			IF arrActualPrioInTurn[3] = 1 AND Lynus_Standards.GVL_Energy.stDataElectricHeatingElements[diNrOfEMS_OUT,liCounterCkeckDeviceAndPrio].byPriority = 1 AND
				(Lynus_Standards.GVL_Energy.stDataElectricHeatingElements[diNrOfEMS_OUT,liCounterCkeckDeviceAndPrio].arrTargetPowerEMS[1] <> 0 OR Lynus_Standards.GVL_Energy.stDataElectricHeatingElements[diNrOfEMS_OUT,liCounterCkeckDeviceAndPrio].arrTargetPowerEMS[2] <> 0 OR
					Lynus_Standards.GVL_Energy.stDataElectricHeatingElements[diNrOfEMS_OUT,liCounterCkeckDeviceAndPrio].arrTargetPowerEMS[3] <> 0 OR Lynus_Standards.GVL_Energy.stDataElectricHeatingElements[diNrOfEMS_OUT,liCounterCkeckDeviceAndPrio].arrTargetPowerEMS[4] <> 0 OR
						Lynus_Standards.GVL_Energy.stDataElectricHeatingElements[diNrOfEMS_OUT,liCounterCkeckDeviceAndPrio].arrTargetPowerEMS[5] <> 0 OR Lynus_Standards.GVL_Energy.stDataElectricHeatingElements[diNrOfEMS_OUT,liCounterCkeckDeviceAndPrio].arrTargetPowerEMS[6] <> 0 OR
							Lynus_Standards.GVL_Energy.stDataElectricHeatingElements[diNrOfEMS_OUT,liCounterCkeckDeviceAndPrio].arrTargetPowerEMS[7] <> 0 OR Lynus_Standards.GVL_Energy.stDataElectricHeatingElements[diNrOfEMS_OUT,liCounterCkeckDeviceAndPrio].arrTargetPowerEMS[8] <> 0 OR
								Lynus_Standards.GVL_Energy.stDataElectricHeatingElements[diNrOfEMS_OUT,liCounterCkeckDeviceAndPrio].arrTargetPowerEMS[9] <> 0 OR Lynus_Standards.GVL_Energy.stDataElectricHeatingElements[diNrOfEMS_OUT,liCounterCkeckDeviceAndPrio].arrTargetPowerEMS[10] <> 0) THEN 
									liNrOfNotDoneDevices := liNrOfNotDoneDevices + 1; 
			END_IF
				//1 Step
				IF arrActualPrioInTurn[3] = 255 AND Lynus_Standards.GVL_Energy.stDataElectricHeatingElements[diNrOfEMS_OUT,liCounterCkeckDeviceAndPrio].byPriority = 255 AND Lynus_Standards.GVL_Energy.stDataElectricHeatingElements[diNrOfEMS_OUT,liCounterCkeckDeviceAndPrio].byNumberOfSteps = 1 AND 
					Lynus_Standards.GVL_Energy.stDataElectricHeatingElements[diNrOfEMS_OUT,liCounterCkeckDeviceAndPrio].arrTargetPowerEMS[1] < 100 THEN 
						liNrOfNotDoneDevices := liNrOfNotDoneDevices + 1; 
				//2 Steps
				ELSIF arrActualPrioInTurn[3] = 255 AND Lynus_Standards.GVL_Energy.stDataElectricHeatingElements[diNrOfEMS_OUT,liCounterCkeckDeviceAndPrio].byPriority = 255 AND Lynus_Standards.GVL_Energy.stDataElectricHeatingElements[diNrOfEMS_OUT,liCounterCkeckDeviceAndPrio].byNumberOfSteps = 2 AND 
					(Lynus_Standards.GVL_Energy.stDataElectricHeatingElements[diNrOfEMS_OUT,liCounterCkeckDeviceAndPrio].arrTargetPowerEMS[1] < 100 OR Lynus_Standards.GVL_Energy.stDataElectricHeatingElements[diNrOfEMS_OUT,liCounterCkeckDeviceAndPrio].arrTargetPowerEMS[2] < 100) THEN 
						liNrOfNotDoneDevices := liNrOfNotDoneDevices + 1; 
				//3 Steps
				ELSIF arrActualPrioInTurn[3] = 255 AND Lynus_Standards.GVL_Energy.stDataElectricHeatingElements[diNrOfEMS_OUT,liCounterCkeckDeviceAndPrio].byPriority = 255 AND Lynus_Standards.GVL_Energy.stDataElectricHeatingElements[diNrOfEMS_OUT,liCounterCkeckDeviceAndPrio].byNumberOfSteps = 3 AND 
					(Lynus_Standards.GVL_Energy.stDataElectricHeatingElements[diNrOfEMS_OUT,liCounterCkeckDeviceAndPrio].arrTargetPowerEMS[1] < 100 OR Lynus_Standards.GVL_Energy.stDataElectricHeatingElements[diNrOfEMS_OUT,liCounterCkeckDeviceAndPrio].arrTargetPowerEMS[2] < 100 OR
						Lynus_Standards.GVL_Energy.stDataElectricHeatingElements[diNrOfEMS_OUT,liCounterCkeckDeviceAndPrio].arrTargetPowerEMS[3] < 100) THEN 
							liNrOfNotDoneDevices := liNrOfNotDoneDevices + 1;
				//4 Steps
				ELSIF arrActualPrioInTurn[3] = 255 AND Lynus_Standards.GVL_Energy.stDataElectricHeatingElements[diNrOfEMS_OUT,liCounterCkeckDeviceAndPrio].byPriority = 255 AND Lynus_Standards.GVL_Energy.stDataElectricHeatingElements[diNrOfEMS_OUT,liCounterCkeckDeviceAndPrio].byNumberOfSteps = 4 AND 
					(Lynus_Standards.GVL_Energy.stDataElectricHeatingElements[diNrOfEMS_OUT,liCounterCkeckDeviceAndPrio].arrTargetPowerEMS[1] < 100 OR Lynus_Standards.GVL_Energy.stDataElectricHeatingElements[diNrOfEMS_OUT,liCounterCkeckDeviceAndPrio].arrTargetPowerEMS[2] < 100 OR
						Lynus_Standards.GVL_Energy.stDataElectricHeatingElements[diNrOfEMS_OUT,liCounterCkeckDeviceAndPrio].arrTargetPowerEMS[3] < 100 OR Lynus_Standards.GVL_Energy.stDataElectricHeatingElements[diNrOfEMS_OUT,liCounterCkeckDeviceAndPrio].arrTargetPowerEMS[4] < 100) THEN 
							liNrOfNotDoneDevices := liNrOfNotDoneDevices + 1;  
				//5 Steps
				ELSIF arrActualPrioInTurn[3] = 255 AND Lynus_Standards.GVL_Energy.stDataElectricHeatingElements[diNrOfEMS_OUT,liCounterCkeckDeviceAndPrio].byPriority = 255 AND Lynus_Standards.GVL_Energy.stDataElectricHeatingElements[diNrOfEMS_OUT,liCounterCkeckDeviceAndPrio].byNumberOfSteps = 5 AND 
					(Lynus_Standards.GVL_Energy.stDataElectricHeatingElements[diNrOfEMS_OUT,liCounterCkeckDeviceAndPrio].arrTargetPowerEMS[1] < 100 OR Lynus_Standards.GVL_Energy.stDataElectricHeatingElements[diNrOfEMS_OUT,liCounterCkeckDeviceAndPrio].arrTargetPowerEMS[2] < 100 OR
						Lynus_Standards.GVL_Energy.stDataElectricHeatingElements[diNrOfEMS_OUT,liCounterCkeckDeviceAndPrio].arrTargetPowerEMS[3] < 100 OR Lynus_Standards.GVL_Energy.stDataElectricHeatingElements[diNrOfEMS_OUT,liCounterCkeckDeviceAndPrio].arrTargetPowerEMS[4] < 100 OR
							Lynus_Standards.GVL_Energy.stDataElectricHeatingElements[diNrOfEMS_OUT,liCounterCkeckDeviceAndPrio].arrTargetPowerEMS[5] < 100) THEN 
								liNrOfNotDoneDevices := liNrOfNotDoneDevices + 1; 
				//6 Steps
				ELSIF arrActualPrioInTurn[3] = 255 AND Lynus_Standards.GVL_Energy.stDataElectricHeatingElements[diNrOfEMS_OUT,liCounterCkeckDeviceAndPrio].byPriority = 255 AND Lynus_Standards.GVL_Energy.stDataElectricHeatingElements[diNrOfEMS_OUT,liCounterCkeckDeviceAndPrio].byNumberOfSteps = 6 AND 
					(Lynus_Standards.GVL_Energy.stDataElectricHeatingElements[diNrOfEMS_OUT,liCounterCkeckDeviceAndPrio].arrTargetPowerEMS[1] < 100 OR Lynus_Standards.GVL_Energy.stDataElectricHeatingElements[diNrOfEMS_OUT,liCounterCkeckDeviceAndPrio].arrTargetPowerEMS[2] < 100 OR
						Lynus_Standards.GVL_Energy.stDataElectricHeatingElements[diNrOfEMS_OUT,liCounterCkeckDeviceAndPrio].arrTargetPowerEMS[3] < 100 OR Lynus_Standards.GVL_Energy.stDataElectricHeatingElements[diNrOfEMS_OUT,liCounterCkeckDeviceAndPrio].arrTargetPowerEMS[4] < 100 OR
							Lynus_Standards.GVL_Energy.stDataElectricHeatingElements[diNrOfEMS_OUT,liCounterCkeckDeviceAndPrio].arrTargetPowerEMS[5] < 100 OR Lynus_Standards.GVL_Energy.stDataElectricHeatingElements[diNrOfEMS_OUT,liCounterCkeckDeviceAndPrio].arrTargetPowerEMS[6] < 100) THEN 
								liNrOfNotDoneDevices := liNrOfNotDoneDevices + 1; 
				//7 Steps
				ELSIF arrActualPrioInTurn[3] = 255 AND Lynus_Standards.GVL_Energy.stDataElectricHeatingElements[diNrOfEMS_OUT,liCounterCkeckDeviceAndPrio].byPriority = 255 AND Lynus_Standards.GVL_Energy.stDataElectricHeatingElements[diNrOfEMS_OUT,liCounterCkeckDeviceAndPrio].byNumberOfSteps = 7 AND 
					(Lynus_Standards.GVL_Energy.stDataElectricHeatingElements[diNrOfEMS_OUT,liCounterCkeckDeviceAndPrio].arrTargetPowerEMS[1] < 100 OR Lynus_Standards.GVL_Energy.stDataElectricHeatingElements[diNrOfEMS_OUT,liCounterCkeckDeviceAndPrio].arrTargetPowerEMS[2] < 100 OR
						Lynus_Standards.GVL_Energy.stDataElectricHeatingElements[diNrOfEMS_OUT,liCounterCkeckDeviceAndPrio].arrTargetPowerEMS[3] < 100 OR Lynus_Standards.GVL_Energy.stDataElectricHeatingElements[diNrOfEMS_OUT,liCounterCkeckDeviceAndPrio].arrTargetPowerEMS[4] < 100 OR
							Lynus_Standards.GVL_Energy.stDataElectricHeatingElements[diNrOfEMS_OUT,liCounterCkeckDeviceAndPrio].arrTargetPowerEMS[5] < 100 OR Lynus_Standards.GVL_Energy.stDataElectricHeatingElements[diNrOfEMS_OUT,liCounterCkeckDeviceAndPrio].arrTargetPowerEMS[6] < 100 OR
								Lynus_Standards.GVL_Energy.stDataElectricHeatingElements[diNrOfEMS_OUT,liCounterCkeckDeviceAndPrio].arrTargetPowerEMS[7] < 100) THEN 
									liNrOfNotDoneDevices := liNrOfNotDoneDevices + 1; 
				//8 Steps
				ELSIF arrActualPrioInTurn[3] = 255 AND Lynus_Standards.GVL_Energy.stDataElectricHeatingElements[diNrOfEMS_OUT,liCounterCkeckDeviceAndPrio].byPriority = 255 AND Lynus_Standards.GVL_Energy.stDataElectricHeatingElements[diNrOfEMS_OUT,liCounterCkeckDeviceAndPrio].byNumberOfSteps = 8 AND 
					(Lynus_Standards.GVL_Energy.stDataElectricHeatingElements[diNrOfEMS_OUT,liCounterCkeckDeviceAndPrio].arrTargetPowerEMS[1] < 100 OR Lynus_Standards.GVL_Energy.stDataElectricHeatingElements[diNrOfEMS_OUT,liCounterCkeckDeviceAndPrio].arrTargetPowerEMS[2] < 100 OR
						Lynus_Standards.GVL_Energy.stDataElectricHeatingElements[diNrOfEMS_OUT,liCounterCkeckDeviceAndPrio].arrTargetPowerEMS[3] < 100 OR Lynus_Standards.GVL_Energy.stDataElectricHeatingElements[diNrOfEMS_OUT,liCounterCkeckDeviceAndPrio].arrTargetPowerEMS[4] < 100 OR
							Lynus_Standards.GVL_Energy.stDataElectricHeatingElements[diNrOfEMS_OUT,liCounterCkeckDeviceAndPrio].arrTargetPowerEMS[5] < 100 OR Lynus_Standards.GVL_Energy.stDataElectricHeatingElements[diNrOfEMS_OUT,liCounterCkeckDeviceAndPrio].arrTargetPowerEMS[6] < 100 OR
								Lynus_Standards.GVL_Energy.stDataElectricHeatingElements[diNrOfEMS_OUT,liCounterCkeckDeviceAndPrio].arrTargetPowerEMS[7] < 100 OR Lynus_Standards.GVL_Energy.stDataElectricHeatingElements[diNrOfEMS_OUT,liCounterCkeckDeviceAndPrio].arrTargetPowerEMS[8] < 100) THEN 
									liNrOfNotDoneDevices := liNrOfNotDoneDevices + 1; 
				//9 Steps
				ELSIF arrActualPrioInTurn[3] = 255 AND Lynus_Standards.GVL_Energy.stDataElectricHeatingElements[diNrOfEMS_OUT,liCounterCkeckDeviceAndPrio].byPriority = 255 AND Lynus_Standards.GVL_Energy.stDataElectricHeatingElements[diNrOfEMS_OUT,liCounterCkeckDeviceAndPrio].byNumberOfSteps = 9 AND 
					(Lynus_Standards.GVL_Energy.stDataElectricHeatingElements[diNrOfEMS_OUT,liCounterCkeckDeviceAndPrio].arrTargetPowerEMS[1] < 100 OR Lynus_Standards.GVL_Energy.stDataElectricHeatingElements[diNrOfEMS_OUT,liCounterCkeckDeviceAndPrio].arrTargetPowerEMS[2] < 100 OR
						Lynus_Standards.GVL_Energy.stDataElectricHeatingElements[diNrOfEMS_OUT,liCounterCkeckDeviceAndPrio].arrTargetPowerEMS[3] < 100 OR Lynus_Standards.GVL_Energy.stDataElectricHeatingElements[diNrOfEMS_OUT,liCounterCkeckDeviceAndPrio].arrTargetPowerEMS[4] < 100 OR
							Lynus_Standards.GVL_Energy.stDataElectricHeatingElements[diNrOfEMS_OUT,liCounterCkeckDeviceAndPrio].arrTargetPowerEMS[5] < 100 OR Lynus_Standards.GVL_Energy.stDataElectricHeatingElements[diNrOfEMS_OUT,liCounterCkeckDeviceAndPrio].arrTargetPowerEMS[6] < 100 OR
								Lynus_Standards.GVL_Energy.stDataElectricHeatingElements[diNrOfEMS_OUT,liCounterCkeckDeviceAndPrio].arrTargetPowerEMS[7] < 100 OR Lynus_Standards.GVL_Energy.stDataElectricHeatingElements[diNrOfEMS_OUT,liCounterCkeckDeviceAndPrio].arrTargetPowerEMS[8] < 100 OR
									Lynus_Standards.GVL_Energy.stDataElectricHeatingElements[diNrOfEMS_OUT,liCounterCkeckDeviceAndPrio].arrTargetPowerEMS[9] < 100) THEN 
										liNrOfNotDoneDevices := liNrOfNotDoneDevices + 1; 
				//10 Steps
				ELSIF arrActualPrioInTurn[3] = 255 AND Lynus_Standards.GVL_Energy.stDataElectricHeatingElements[diNrOfEMS_OUT,liCounterCkeckDeviceAndPrio].byPriority = 255 AND Lynus_Standards.GVL_Energy.stDataElectricHeatingElements[diNrOfEMS_OUT,liCounterCkeckDeviceAndPrio].byNumberOfSteps = 10 AND 
					(Lynus_Standards.GVL_Energy.stDataElectricHeatingElements[diNrOfEMS_OUT,liCounterCkeckDeviceAndPrio].arrTargetPowerEMS[1] < 100 OR Lynus_Standards.GVL_Energy.stDataElectricHeatingElements[diNrOfEMS_OUT,liCounterCkeckDeviceAndPrio].arrTargetPowerEMS[2] < 100 OR
						Lynus_Standards.GVL_Energy.stDataElectricHeatingElements[diNrOfEMS_OUT,liCounterCkeckDeviceAndPrio].arrTargetPowerEMS[3] < 100 OR Lynus_Standards.GVL_Energy.stDataElectricHeatingElements[diNrOfEMS_OUT,liCounterCkeckDeviceAndPrio].arrTargetPowerEMS[4] < 100 OR
							Lynus_Standards.GVL_Energy.stDataElectricHeatingElements[diNrOfEMS_OUT,liCounterCkeckDeviceAndPrio].arrTargetPowerEMS[5] < 100 OR Lynus_Standards.GVL_Energy.stDataElectricHeatingElements[diNrOfEMS_OUT,liCounterCkeckDeviceAndPrio].arrTargetPowerEMS[6] < 100 OR
								Lynus_Standards.GVL_Energy.stDataElectricHeatingElements[diNrOfEMS_OUT,liCounterCkeckDeviceAndPrio].arrTargetPowerEMS[7] < 100 OR Lynus_Standards.GVL_Energy.stDataElectricHeatingElements[diNrOfEMS_OUT,liCounterCkeckDeviceAndPrio].arrTargetPowerEMS[8] < 100 OR
									Lynus_Standards.GVL_Energy.stDataElectricHeatingElements[diNrOfEMS_OUT,liCounterCkeckDeviceAndPrio].arrTargetPowerEMS[9] < 100 OR Lynus_Standards.GVL_Energy.stDataElectricHeatingElements[diNrOfEMS_OUT,liCounterCkeckDeviceAndPrio].arrTargetPowerEMS[10] < 100) THEN 
										liNrOfNotDoneDevices := liNrOfNotDoneDevices + 1; 
				END_IF
		
		IF arrActualPrioInTurn[3] = 1 AND uiState = 70 AND liNrOfNotDoneDevices = 0 AND arrCTCheckActivePrio[3] = Constants_Energy.diMaxNumberOfElectricHeatingElements AND liCounterCkeckDeviceAndPrio = Constants_Energy.diMaxNumberOfElectricHeatingElements THEN 
			arrMinPrioReached[3] := TRUE; arrMaxPrioReached[3] := FALSE; liNrOfNotDoneDevices := 0; uiState := 90; arrCTCheckActivePrio[3] := 0; liCounterCkeckDeviceAndPrio := 0; 
		END_IF
		IF arrActualPrioInTurn[3] = 255 AND uiState = 70 AND liNrOfNotDoneDevices = 0 AND arrCTCheckActivePrio[3] = Constants_Energy.diMaxNumberOfElectricHeatingElements AND liCounterCkeckDeviceAndPrio = Constants_Energy.diMaxNumberOfElectricHeatingElements THEN 
			arrMaxPrioReached[3] := TRUE; arrMinPrioReached[3] := FALSE; liNrOfNotDoneDevices := 0; uiState := 90; arrCTCheckActivePrio[3] := 0; liCounterCkeckDeviceAndPrio := 0; 
		END_IF
		
		//Timout, go to next step
		IF timTimeout.Q AND uiState = 70 THEN uiState := 90; END_IF
		
	90: //Check the priority for the big consumer to controll it
		uiState_CP := uiState;
	
		//First check if we have min 1 of this Device Type. If not, complete this Device Type and go to the next step
		//Check also the bigest Priority of this Device Type
		diNumberOfDevicesFromEachType := 0; bySearchBigestPrio := 0;
		FOR liLPCheckDeviceAndPrio := 1 TO Constants_Energy.diMaxNumberOfOtherBigConsumers BY 1 DO
			IF Lynus_Standards.GVL_Energy.stDataOtherBigConsumers[diNrOfEMS_OUT,liLPCheckDeviceAndPrio].byPriority <> 0 THEN diNumberOfDevicesFromEachType := diNumberOfDevicesFromEachType + 1; END_IF
				IF Lynus_Standards.GVL_Energy.stDataOtherBigConsumers[diNrOfEMS_OUT,liLPCheckDeviceAndPrio].byPriority > bySearchBigestPrio THEN bySearchBigestPrio := Lynus_Standards.GVL_Energy.stDataOtherBigConsumers[diNrOfEMS_OUT,liLPCheckDeviceAndPrio].byPriority; END_IF   
		END_FOR 
			IF bSurplusAvailable AND arrActualPrioInTurn[4] > bySearchBigestPrio AND uiState = 90 THEN arrActualPrioInTurn[4] := 255; END_IF
				IF NOT bSurplusAvailable AND arrActualPrioInTurn[4] > bySearchBigestPrio AND uiState = 90 THEN arrActualPrioInTurn[4] := bySearchBigestPrio; END_IF
		
			IF bSurplusAvailable AND diNumberOfDevicesFromEachType = 0 THEN arrActualPrioInTurn[4] := 255; END_IF
				IF NOT bSurplusAvailable AND diNumberOfDevicesFromEachType = 0 THEN arrActualPrioInTurn[4] := 1; END_IF
		
		//Count up each Device
		arrCTCheckActivePrio[4] := arrCTCheckActivePrio[4] + 1;
			arrCTCheckActivePrio[4] := LIMIT(1,arrCTCheckActivePrio[4],Constants_Energy.diMaxNumberOfOtherBigConsumers);
		
			//Surplus
			IF bSurplusAvailable AND Lynus_Standards.GVL_Energy.stDataOtherBigConsumers[diNrOfEMS_OUT,arrCTCheckActivePrio[4]].byPriority = arrActualPrioInTurn[4] AND Lynus_Standards.GVL_Energy.stDataOtherBigConsumers[diNrOfEMS_OUT,arrCTCheckActivePrio[4]].rTargetPowerEMS < 100 THEN
				arrMaxPrioReached[4] := FALSE;
					arrMinPrioReached[4] := FALSE;
						arrCTCheckActivePrio[4] := 0;
							uiState := 109; 
			ELSE
				IF bSurplusAvailable AND arrActualPrioInTurn[4] < 255 AND uiState = 90 AND arrCTCheckActivePrio[4] = Constants_Energy.diMaxNumberOfOtherBigConsumers THEN arrActualPrioInTurn[4] := arrActualPrioInTurn[4] + 1; arrCTCheckActivePrio[4] := 0; END_IF
			END_IF
				//No surplus
				IF NOT bSurplusAvailable AND Lynus_Standards.GVL_Energy.stDataOtherBigConsumers[diNrOfEMS_OUT,arrCTCheckActivePrio[4]].byPriority = arrActualPrioInTurn[4] AND Lynus_Standards.GVL_Energy.stDataOtherBigConsumers[diNrOfEMS_OUT,arrCTCheckActivePrio[4]].rTargetPowerEMS > 0 THEN
					arrMaxPrioReached[4] := FALSE;
						arrMinPrioReached[4] := FALSE;
							arrCTCheckActivePrio[4] := 0;
								uiState := 109;
				ELSE
					IF NOT bSurplusAvailable AND arrActualPrioInTurn[4] > 1 AND uiState = 90 AND arrCTCheckActivePrio[4] = Constants_Energy.diMaxNumberOfOtherBigConsumers THEN arrActualPrioInTurn[4] := arrActualPrioInTurn[4] - 1; arrCTCheckActivePrio[4] := 0; END_IF
				END_IF
		
		
		//Go to next step if we are on min prio or on max prio and the target power is just set to the min or to the max value.
		liNrOfNotDoneDevices := 0;
			FOR liLPCheckDeviceAndPrio := 1 TO Constants_Energy.diMaxNumberOfOtherBigConsumers BY 1 DO
				IF arrActualPrioInTurn[4] = 1 AND Lynus_Standards.GVL_Energy.stDataOtherBigConsumers[diNrOfEMS_OUT,liLPCheckDeviceAndPrio].rTargetPowerEMS <> 0 AND Lynus_Standards.GVL_Energy.stDataOtherBigConsumers[diNrOfEMS_OUT,liLPCheckDeviceAndPrio].byPriority = 1 THEN
					liNrOfNotDoneDevices := liNrOfNotDoneDevices + 1;	
				END_IF
					IF arrActualPrioInTurn[4] = 255 AND Lynus_Standards.GVL_Energy.stDataOtherBigConsumers[diNrOfEMS_OUT,liLPCheckDeviceAndPrio].rTargetPowerEMS < 100 AND Lynus_Standards.GVL_Energy.stDataOtherBigConsumers[diNrOfEMS_OUT,liLPCheckDeviceAndPrio].byPriority = 255 THEN
						liNrOfNotDoneDevices := liNrOfNotDoneDevices + 1;	
					END_IF
			END_FOR	
		
		IF arrActualPrioInTurn[4] = 1 AND uiState = 90 AND liNrOfNotDoneDevices = 0 AND arrCTCheckActivePrio[4] = Constants_Energy.diMaxNumberOfOtherBigConsumers THEN 
			arrMinPrioReached[4] := TRUE; arrMaxPrioReached[4] := FALSE; liNrOfNotDoneDevices := 0; uiState := 109; arrCTCheckActivePrio[4] := 0; 
		END_IF
		IF arrActualPrioInTurn[4] = 255 AND uiState = 90 AND liNrOfNotDoneDevices = 0 AND arrCTCheckActivePrio[4] = Constants_Energy.diMaxNumberOfOtherBigConsumers THEN 
			arrMaxPrioReached[4] := TRUE; arrMinPrioReached[4] := FALSE; liNrOfNotDoneDevices := 0; uiState := 109; arrCTCheckActivePrio[4] := 0; 
		END_IF
		
		//Timout, go to next step
		IF timTimeout.Q AND uiState = 90 THEN uiState := 109; END_IF
		
	109://Check if in Load management mode or Peak shaving mode some electric Fuse Line use to much power when we have here surplus
		uiState_CP := uiState;

		//Count up each Device
		arrCTCheckActivePrio[5] := arrCTCheckActivePrio[5] + 1;
			arrCTCheckActivePrio[5] := LIMIT(1,arrCTCheckActivePrio[5],Constants_Energy.diMaxNumberOfElectricChargingStations);
		
		IF ((eOperationMode = E_OperatingMode_EMS.eLoadManagement OR eOperationMode = E_OperatingMode_EMS.ePeakLoadCapping) AND bSurplusAvailable AND stSetupEMS.bEnableMainFuseFunction) THEN
			IF Lynus_Standards.GVL_Energy.stDataElectricChargingStations[diNrOfEMS_OUT,arrCTCheckActivePrio[5]].byPriority = arrActualPrioInTurn[5] THEN
				//The ECS use to much power. So dont give here more power. Go to next priority
				IF bNoPowerForECS THEN
					//Go to next prio that we can go forward with the other Devices with same priority. Controlling for ECS see down on the Part on wich we limit the charging station about the electric Fuse Line
					IF arrActualPrioInTurn[5] < 255 THEN arrActualPrioInTurn[5] := arrActualPrioInTurn[5] + 1; END_IF
						uiState := 110;
							arrCTCheckActivePrio[5] := 0;	
				END_IF
			END_IF 
		ELSE
			uiState := 110;
				arrCTCheckActivePrio[5] := 0;
		END_IF
		
		//Go to next step if wa have checked every ECS without resluts
		IF arrCTCheckActivePrio[5] >= Constants_Energy.diMaxNumberOfElectricChargingStations AND uiState = 109 THEN
			uiState := 110;
				arrCTCheckActivePrio[5] := 0;
		END_IF 
	 	
		//Timout, go to next step
		IF timTimeout.Q AND uiState = 109 THEN uiState := 110; arrCTCheckActivePrio[5] := 0; END_IF	
		
	110: //Check the priority for the electric charging stations to controll it
		uiState_CP := uiState;
	
		//First check if we have min 1 of this Device Type. If not, complete this Device Type and go to the next step
		//Check also the bigest Priority of this Device Type
		diNumberOfDevicesFromEachType := 0; bySearchBigestPrio := 0;
		FOR liLPCheckDeviceAndPrio := 1 TO Constants_Energy.diMaxNumberOfElectricChargingStations BY 1 DO
			IF Lynus_Standards.GVL_Energy.stDataElectricChargingStations[diNrOfEMS_OUT,liLPCheckDeviceAndPrio].byPriority <> 0 THEN diNumberOfDevicesFromEachType := diNumberOfDevicesFromEachType + 1; END_IF
				IF Lynus_Standards.GVL_Energy.stDataElectricChargingStations[diNrOfEMS_OUT,liLPCheckDeviceAndPrio].byPriority > bySearchBigestPrio THEN bySearchBigestPrio := Lynus_Standards.GVL_Energy.stDataElectricChargingStations[diNrOfEMS_OUT,liLPCheckDeviceAndPrio].byPriority; END_IF   
		END_FOR 
			IF bSurplusAvailable AND arrActualPrioInTurn[5] > bySearchBigestPrio AND uiState = 110 THEN arrActualPrioInTurn[5] := 255; END_IF
				IF NOT bSurplusAvailable AND arrActualPrioInTurn[5] > bySearchBigestPrio AND uiState = 110 THEN arrActualPrioInTurn[5] := bySearchBigestPrio; END_IF
		
			IF bSurplusAvailable AND diNumberOfDevicesFromEachType = 0 THEN arrActualPrioInTurn[5] := 255; END_IF
				IF NOT bSurplusAvailable AND diNumberOfDevicesFromEachType = 0 THEN arrActualPrioInTurn[5] := 1; END_IF
		
		//Count up each Device
		arrCTCheckActivePrio[5] := arrCTCheckActivePrio[5] + 1;
			arrCTCheckActivePrio[5] := LIMIT(1,arrCTCheckActivePrio[5],Constants_Energy.diMaxNumberOfElectricChargingStations);
		
			//Surplus
			IF bSurplusAvailable AND Lynus_Standards.GVL_Energy.stDataElectricChargingStations[diNrOfEMS_OUT,arrCTCheckActivePrio[5]].byPriority = arrActualPrioInTurn[5] AND Lynus_Standards.GVL_Energy.stDataElectricChargingStations[diNrOfEMS_OUT,arrCTCheckActivePrio[5]].rTargetPowerEMS < 100 THEN
				arrMaxPrioReached[5] := FALSE;
					arrMinPrioReached[5] := FALSE;
						arrCTCheckActivePrio[5] := 0;
							uiState := 130;
			ELSE
				IF bSurplusAvailable AND arrActualPrioInTurn[5] < 255 AND uiState = 110 AND arrCTCheckActivePrio[5] = Constants_Energy.diMaxNumberOfElectricChargingStations THEN arrActualPrioInTurn[5] := arrActualPrioInTurn[5] + 1; arrCTCheckActivePrio[5] := 0; END_IF
			END_IF
				//No surplus
				IF NOT bSurplusAvailable AND Lynus_Standards.GVL_Energy.stDataElectricChargingStations[diNrOfEMS_OUT,arrCTCheckActivePrio[5]].byPriority = arrActualPrioInTurn[5] AND Lynus_Standards.GVL_Energy.stDataElectricChargingStations[diNrOfEMS_OUT,arrCTCheckActivePrio[5]].rTargetPowerEMS > 0 THEN
					arrMaxPrioReached[5] := FALSE;
						arrMinPrioReached[5] := FALSE;
							arrCTCheckActivePrio[5] := 0;
								uiState := 130;
				ELSE
					IF NOT bSurplusAvailable AND arrActualPrioInTurn[5] > 1 AND uiState = 110 AND arrCTCheckActivePrio[5] = Constants_Energy.diMaxNumberOfElectricChargingStations THEN arrActualPrioInTurn[5] := arrActualPrioInTurn[5] - 1; arrCTCheckActivePrio[5] := 0; END_IF
				END_IF
		
		//Go to next step if we are on min prio or on max prio and the target power is just set to the min or to the max value.
		liNrOfNotDoneDevices := 0;
			FOR liLPCheckDeviceAndPrio := 1 TO Constants_Energy.diMaxNumberOfElectricChargingStations BY 1 DO
				IF arrActualPrioInTurn[5] = 1 AND Lynus_Standards.GVL_Energy.stDataElectricChargingStations[diNrOfEMS_OUT,liLPCheckDeviceAndPrio].rTargetPowerEMS <> 0 AND Lynus_Standards.GVL_Energy.stDataElectricChargingStations[diNrOfEMS_OUT,liLPCheckDeviceAndPrio].byPriority = 1 THEN
					liNrOfNotDoneDevices := liNrOfNotDoneDevices + 1;	
				END_IF
					IF arrActualPrioInTurn[5] = 255 AND Lynus_Standards.GVL_Energy.stDataElectricChargingStations[diNrOfEMS_OUT,liLPCheckDeviceAndPrio].rTargetPowerEMS < 100 AND Lynus_Standards.GVL_Energy.stDataElectricChargingStations[diNrOfEMS_OUT,liLPCheckDeviceAndPrio].byPriority = 255 THEN
						liNrOfNotDoneDevices := liNrOfNotDoneDevices + 1;	
					END_IF
			END_FOR
		
		IF arrActualPrioInTurn[5] = 1 AND uiState = 110 AND liNrOfNotDoneDevices = 0 AND arrCTCheckActivePrio[5] = Constants_Energy.diMaxNumberOfElectricChargingStations THEN 
			arrMinPrioReached[5] := TRUE; arrMaxPrioReached[5] := FALSE; liNrOfNotDoneDevices := 0; uiState := 130; arrCTCheckActivePrio[5] := 0; 
		END_IF
		IF arrActualPrioInTurn[5] = 255 AND uiState = 110 AND liNrOfNotDoneDevices = 0 AND arrCTCheckActivePrio[5] = Constants_Energy.diMaxNumberOfElectricChargingStations THEN 
			arrMaxPrioReached[5] := TRUE; arrMinPrioReached[5] := FALSE; liNrOfNotDoneDevices := 0; uiState := 130; arrCTCheckActivePrio[5] := 0; 
		END_IF	
		
		//Timout, go to next step
		IF timTimeout.Q AND uiState = 110 THEN uiState := 130; END_IF
		
	130: //Search the smallest/biggest common priority and the number of devices with the same priority  
		IF bSurplusAvailable THEN bySmGrActiveCommonPrio := 255; END_IF
		IF NOT bSurplusAvailable THEN bySmGrActiveCommonPrio := 1; END_IF
	
		FOR byLPSmActiveCommonPrio := 1 TO 5 BY 1 DO
			IF bSurplusAvailable AND arrActualPrioInTurn[byLPSmActiveCommonPrio] < bySmGrActiveCommonPrio THEN bySmGrActiveCommonPrio := arrActualPrioInTurn[byLPSmActiveCommonPrio]; END_IF 
			IF NOT bSurplusAvailable AND arrActualPrioInTurn[byLPSmActiveCommonPrio] > bySmGrActiveCommonPrio THEN bySmGrActiveCommonPrio := arrActualPrioInTurn[byLPSmActiveCommonPrio]; END_IF 
		END_FOR
		
		//Back to the start when complete power is awarded, all power is set on 0 or we haven't common priority 	
		IF (arrMaxPrioReached[1] AND arrMaxPrioReached[2] AND arrMaxPrioReached[3] AND arrMaxPrioReached[4] AND arrMaxPrioReached[5]) OR
			(arrMinPrioReached[1] AND arrMinPrioReached[2] AND arrMinPrioReached[3] AND arrMinPrioReached[4] AND arrMinPrioReached[5]) THEN
				uiState := 10;
		ELSE
				uiState := 131;
		END_IF
		
	131: //Ckeck if the Batterys are full or not when we have no surplus. Thus the problem can be avoided if the battery FB regulates the power internally to 0, but the EMS still sends power to the inverter.
		 //Because otherwise it always takes too long when we have a small consumption and the battery must first be regulated to 0% in the GVL, although you are already full and you can therefore no longer be regulated back.
		 
		IF eOperationMode = E_OperatingMode_EMS.eSelfConsumption THEN 
			FOR liLPDataBatteryInverter := 1 TO Constants_Energy.diMaxNumberOfBatteryInverters BY 1 DO
				IF NOT bSurplusAvailable AND Lynus_Standards.GVL_Energy.stDataOfBatteryInverters[diNrOfEMS_OUT,liLPDataBatteryInverter].byPriority = bySmGrActiveCommonPrio AND 
					arrTimBatterysAreFull[liLPDataBatteryInverter].Q THEN
						Lynus_Standards.GVL_Energy.stDataOfBatteryInverters[diNrOfEMS_OUT,liLPDataBatteryInverter].rTargetPowerEMS := 0;
				END_IF	  
			END_FOR 
	
			//When we have a surplus again and the battery is full, we control it again with - 99.99%, so that the following devices do not have to wait too long to be controlled. 	
			//It must be set to 99.99, otherwise an error would occur in the next step.
			FOR liLPDataBatteryInverter := 1 TO Constants_Energy.diMaxNumberOfBatteryInverters BY 1 DO
				IF bSurplusAvailable AND Lynus_Standards.GVL_Energy.stDataOfBatteryInverters[diNrOfEMS_OUT,liLPDataBatteryInverter].byPriority = bySmGrActiveCommonPrio AND 
					arrTimBatterysAreFull[liLPDataBatteryInverter].Q THEN
						Lynus_Standards.GVL_Energy.stDataOfBatteryInverters[diNrOfEMS_OUT,liLPDataBatteryInverter].rTargetPowerEMS := - 99.99;
				END_IF	  
			END_FOR
		END_IF
		
		//Go to the next Step
		uiState := 150;
		
	150: //Calcualte the % power from each device with the same priority
		lrMaxPowerDevicesWithActualPrio := 0;
			bMissingPowerData := FALSE;
		
		//Batterys are only a "normal" Device, when the self consumption mode is active.
		IF eOperationMode = E_OperatingMode_EMS.eSelfConsumption THEN 
			//Batteryinverters
			FOR liLPCheckMaxPower := 1 TO Constants_Energy.diMaxNumberOfBatteryInverters BY 1 DO
				IF bSurplusAvailable AND Lynus_Standards.GVL_Energy.stDataOfBatteryInverters[diNrOfEMS_OUT,liLPCheckMaxPower].byPriority = bySmGrActiveCommonPrio AND Lynus_Standards.GVL_Energy.stDataOfBatteryInverters[diNrOfEMS_OUT,liLPCheckMaxPower].rTargetPowerEMS > -100 AND NOT Lynus_Standards.GVL_Energy.stDataOfBatteryInverters[diNrOfEMS_OUT,liLPCheckMaxPower].bWorkOnIslandMode THEN lrMaxPowerDevicesWithActualPrio := lrMaxPowerDevicesWithActualPrio + Lynus_Standards.GVL_Energy.stDataOfBatteryInverters[diNrOfEMS_OUT,liLPCheckMaxPower].rMaxChargePower; END_IF
				IF NOT bSurplusAvailable AND Lynus_Standards.GVL_Energy.stDataOfBatteryInverters[diNrOfEMS_OUT,liLPCheckMaxPower].byPriority = bySmGrActiveCommonPrio AND Lynus_Standards.GVL_Energy.stDataOfBatteryInverters[diNrOfEMS_OUT,liLPCheckMaxPower].rTargetPowerEMS < 0 AND NOT Lynus_Standards.GVL_Energy.stDataOfBatteryInverters[diNrOfEMS_OUT,liLPCheckMaxPower].bWorkOnIslandMode THEN lrMaxPowerDevicesWithActualPrio := lrMaxPowerDevicesWithActualPrio + Lynus_Standards.GVL_Energy.stDataOfBatteryInverters[diNrOfEMS_OUT,liLPCheckMaxPower].rMaxChargePower; END_IF 
			END_FOR
		END_IF
			//Heating pumps
			IF arrActualStepInTurn[1] >= 1 AND arrActualStepInTurn[1] <= 2 THEN
				FOR liLPCheckMaxPower := 1 TO Constants_Energy.diMaxNumberOfHeatingPumps BY 1 DO
					IF bSurplusAvailable AND Lynus_Standards.GVL_Energy.stDataHeatingPumps[diNrOfEMS_OUT,liLPCheckMaxPower].byPriority = bySmGrActiveCommonPrio AND Lynus_Standards.GVL_Energy.stDataHeatingPumps[diNrOfEMS_OUT,liLPCheckMaxPower].arrTargetPowerEMS[arrActualStepInTurn[1]] < 100 THEN lrMaxPowerDevicesWithActualPrio := lrMaxPowerDevicesWithActualPrio + Lynus_Standards.GVL_Energy.stDataHeatingPumps[diNrOfEMS_OUT,liLPCheckMaxPower].arrMaxPower[arrActualStepInTurn[1]]; END_IF
					IF NOT bSurplusAvailable AND Lynus_Standards.GVL_Energy.stDataHeatingPumps[diNrOfEMS_OUT,liLPCheckMaxPower].byPriority = bySmGrActiveCommonPrio AND Lynus_Standards.GVL_Energy.stDataHeatingPumps[diNrOfEMS_OUT,liLPCheckMaxPower].arrTargetPowerEMS[arrActualStepInTurn[1]] > 0 THEN lrMaxPowerDevicesWithActualPrio := lrMaxPowerDevicesWithActualPrio + Lynus_Standards.GVL_Energy.stDataHeatingPumps[diNrOfEMS_OUT,liLPCheckMaxPower].arrMaxPower[arrActualStepInTurn[1]]; END_IF
				END_FOR
			END_IF
				//Electric heating elements
				IF arrActualStepInTurn[2] >= 1 AND arrActualStepInTurn[2] <= 10 THEN
					FOR liLPCheckMaxPower := 1 TO Constants_Energy.diMaxNumberOfElectricHeatingElements BY 1 DO
						IF bSurplusAvailable AND Lynus_Standards.GVL_Energy.stDataElectricHeatingElements[diNrOfEMS_OUT,liLPCheckMaxPower].byPriority = bySmGrActiveCommonPrio AND Lynus_Standards.GVL_Energy.stDataElectricHeatingElements[diNrOfEMS_OUT,liLPCheckMaxPower].arrTargetPowerEMS[arrActualStepInTurn[2]] < 100 THEN lrMaxPowerDevicesWithActualPrio := lrMaxPowerDevicesWithActualPrio + Lynus_Standards.GVL_Energy.stDataElectricHeatingElements[diNrOfEMS_OUT,liLPCheckMaxPower].arrMaxPower[arrActualStepInTurn[2]]; END_IF 
						IF NOT bSurplusAvailable AND Lynus_Standards.GVL_Energy.stDataElectricHeatingElements[diNrOfEMS_OUT,liLPCheckMaxPower].byPriority = bySmGrActiveCommonPrio AND Lynus_Standards.GVL_Energy.stDataElectricHeatingElements[diNrOfEMS_OUT,liLPCheckMaxPower].arrTargetPowerEMS[arrActualStepInTurn[2]] > 0 THEN lrMaxPowerDevicesWithActualPrio := lrMaxPowerDevicesWithActualPrio + Lynus_Standards.GVL_Energy.stDataElectricHeatingElements[diNrOfEMS_OUT,liLPCheckMaxPower].arrMaxPower[arrActualStepInTurn[2]]; END_IF 
					END_FOR	
				END_IF
					//Other big consumer
					FOR liLPCheckMaxPower := 1 TO Constants_Energy.diMaxNumberOfOtherBigConsumers BY 1 DO
						IF bSurplusAvailable AND Lynus_Standards.GVL_Energy.stDataOtherBigConsumers[diNrOfEMS_OUT,liLPCheckMaxPower].byPriority = bySmGrActiveCommonPrio AND Lynus_Standards.GVL_Energy.stDataOtherBigConsumers[diNrOfEMS_OUT,liLPCheckMaxPower].rTargetPowerEMS < 100 THEN lrMaxPowerDevicesWithActualPrio := lrMaxPowerDevicesWithActualPrio + Lynus_Standards.GVL_Energy.stDataOtherBigConsumers[diNrOfEMS_OUT,liLPCheckMaxPower].rMaxPower; END_IF
						IF NOT bSurplusAvailable AND Lynus_Standards.GVL_Energy.stDataOtherBigConsumers[diNrOfEMS_OUT,liLPCheckMaxPower].byPriority = bySmGrActiveCommonPrio AND Lynus_Standards.GVL_Energy.stDataOtherBigConsumers[diNrOfEMS_OUT,liLPCheckMaxPower].rTargetPowerEMS > 0 THEN lrMaxPowerDevicesWithActualPrio := lrMaxPowerDevicesWithActualPrio + Lynus_Standards.GVL_Energy.stDataOtherBigConsumers[diNrOfEMS_OUT,liLPCheckMaxPower].rMaxPower; END_IF
					END_FOR
						//Electric charging stations
						FOR liLPCheckMaxPower := 1 TO Constants_Energy.diMaxNumberOfElectricChargingStations BY 1 DO
							IF bSurplusAvailable AND Lynus_Standards.GVL_Energy.stDataElectricChargingStations[diNrOfEMS_OUT,liLPCheckMaxPower].byPriority = bySmGrActiveCommonPrio AND Lynus_Standards.GVL_Energy.stDataElectricChargingStations[diNrOfEMS_OUT,liLPCheckMaxPower].rTargetPowerEMS < 100 THEN lrMaxPowerDevicesWithActualPrio := lrMaxPowerDevicesWithActualPrio + Lynus_Standards.GVL_Energy.stDataElectricChargingStations[diNrOfEMS_OUT,liLPCheckMaxPower].rMaxPower; END_IF
							IF NOT bSurplusAvailable AND Lynus_Standards.GVL_Energy.stDataElectricChargingStations[diNrOfEMS_OUT,liLPCheckMaxPower].byPriority = bySmGrActiveCommonPrio AND Lynus_Standards.GVL_Energy.stDataElectricChargingStations[diNrOfEMS_OUT,liLPCheckMaxPower].rTargetPowerEMS > 0 THEN lrMaxPowerDevicesWithActualPrio := lrMaxPowerDevicesWithActualPrio + Lynus_Standards.GVL_Energy.stDataElectricChargingStations[diNrOfEMS_OUT,liLPCheckMaxPower].rMaxPower; END_IF 
						END_FOR
		
		//Check is somthing has changed at the actual priority or at the actual step 
		//Priority or step now is higher as before
		IF (bSurplusAvailable AND MEMCMP(ADR(bySmGrActiveCommonPrio),ADR(bySmGrActiveCommonPrio_CP),SIZEOF(bySmGrActiveCommonPrio_CP)) <> 0) OR (bSurplusAvailable AND MEMCMP(ADR(arrActualStepInTurn),ADR(arrActualStepInTurn_CP),SIZEOF(arrActualStepInTurn_CP)) <> 0) THEN
			bySmGrActiveCommonPrio_CP := bySmGrActiveCommonPrio;
				arrActualStepInTurn_CP := arrActualStepInTurn;
					bStepWasOn100 := FALSE;		
		END_IF
			//Priority or step now is lower as before
			IF (NOT bSurplusAvailable AND MEMCMP(ADR(bySmGrActiveCommonPrio),ADR(bySmGrActiveCommonPrio_CP),SIZEOF(bySmGrActiveCommonPrio_CP)) <> 0) OR (NOT bSurplusAvailable AND MEMCMP(ADR(arrActualStepInTurn),ADR(arrActualStepInTurn_CP),SIZEOF(arrActualStepInTurn_CP)) <> 0) THEN
				bySmGrActiveCommonPrio_CP := bySmGrActiveCommonPrio;
					arrActualStepInTurn_CP := arrActualStepInTurn;
						bStepWasOn100 := TRUE;			
			END_IF						
						
		IF lrMaxPowerDevicesWithActualPrio > 0 THEN
			//Calcualte the power for the controllable devices
			IF bSurplusAvailable THEN rValuePercentToControllableDevices := LREAL_TO_REAL((100 * (lrActualSurplusOrConsumption * - 1)) / lrMaxPowerDevicesWithActualPrio); END_IF
  			IF NOT bSurplusAvailable THEN rValuePercentToControllableDevices := LREAL_TO_REAL((100 * lrActualSurplusOrConsumption) / lrMaxPowerDevicesWithActualPrio); END_IF
			//Calcualte the power for the On/Off or step switched devices
			IF bSurplusAvailable THEN rValuePercentToStepSwitchedDevices := LREAL_TO_REAL((100 * (lrActualSurplusOrConsumption * - 1)) / lrMaxPowerDevicesWithActualPrio); END_IF
			IF NOT bSurplusAvailable THEN rValuePercentToStepSwitchedDevices := (100 - LREAL_TO_REAL((100 * lrActualSurplusOrConsumption) / lrMaxPowerDevicesWithActualPrio)); END_IF
				IF bSurplusAvailable AND rValuePercentToStepSwitchedDevices >= 100 THEN bStepWasOn100 := TRUE; END_IF
				IF NOT bSurplusAvailable AND rValuePercentToStepSwitchedDevices < Constants_Energy.byTargetOffPowerForOnOffDevices THEN bStepWasOn100 := FALSE; END_IF
					IF bStepWasOn100 THEN rValuePercentToStepSwitchedDevices := 100; END_IF
					IF NOT bStepWasOn100 THEN rValuePercentToStepSwitchedDevices := 0; END_IF		
		ELSE
			//Power inputs from the setups of the devices are missing. Set the target power automatically to 0
			bMissingPowerData := TRUE;
			IF bSurplusAvailable THEN
				rValuePercentToControllableDevices := - 100;
				rValuePercentToStepSwitchedDevices := 0;
			END_IF
				IF NOT bSurplusAvailable THEN
					rValuePercentToControllableDevices := 100;
					rValuePercentToStepSwitchedDevices := 0;
				END_IF
		END_IF
		
		//If we have more surplus than the maximum power of the devices is, then we can set the target power directly to 100%
		IF bSurplusAvailable AND (lrActualSurplusOrConsumption * - 1) >= lrMaxPowerDevicesWithActualPrio AND NOT bMissingPowerData THEN rValuePercentToControllableDevices := 100; END_IF
		IF bSurplusAvailable AND (lrActualSurplusOrConsumption * - 1) >= lrMaxPowerDevicesWithActualPrio AND NOT bMissingPowerData THEN rValuePercentToStepSwitchedDevices := 100; bStepWasOn100 := TRUE; END_IF
		
		//If more power is consumed than the maximum power of the devices, 0% power can be commanded (for controllable devices 100% as it is deducted).
		IF NOT bSurplusAvailable AND lrActualSurplusOrConsumption >= lrMaxPowerDevicesWithActualPrio AND NOT bMissingPowerData THEN rValuePercentToControllableDevices := 100; END_IF
		IF NOT bSurplusAvailable AND lrActualSurplusOrConsumption >= lrMaxPowerDevicesWithActualPrio AND NOT bMissingPowerData THEN rValuePercentToStepSwitchedDevices := 0; bStepWasOn100 := FALSE; END_IF
		
		//Check the limits
		rValuePercentToControllableDevices := LIMIT(0,rValuePercentToControllableDevices,100);
			rValuePercentToStepSwitchedDevices := LIMIT(0,rValuePercentToStepSwitchedDevices,100);
				
		uiState := 170;
		
	170: //Set the target power to each device
		//Batterys or battery inverters
		//Batterys are only a "normal" Device, when the self consumption mode is active.
		IF eOperationMode = E_OperatingMode_EMS.eSelfConsumption THEN 
			FOR liLPSetPercentPower := 1 TO Constants_Energy.diMaxNumberOfBatteryInverters BY 1 DO
				IF bSurplusAvailable AND Lynus_Standards.GVL_Energy.stDataOfBatteryInverters[diNrOfEMS_OUT,liLPSetPercentPower].byPriority = bySmGrActiveCommonPrio AND Lynus_Standards.GVL_Energy.stDataOfBatteryInverters[diNrOfEMS_OUT,liLPSetPercentPower].rTargetPowerEMS > -100 THEN 
					Lynus_Standards.GVL_Energy.stDataOfBatteryInverters[diNrOfEMS_OUT,liLPSetPercentPower].rTargetPowerEMS := Lynus_Standards.GVL_Energy.stDataOfBatteryInverters[diNrOfEMS_OUT,liLPSetPercentPower].rTargetPowerEMS - rValuePercentToControllableDevices; 
				END_IF
				IF bSurplusAvailable AND Lynus_Standards.GVL_Energy.stDataOfBatteryInverters[diNrOfEMS_OUT,liLPSetPercentPower].rTargetPowerEMS < -100 THEN 
					Lynus_Standards.GVL_Energy.stDataOfBatteryInverters[diNrOfEMS_OUT,liLPSetPercentPower].rTargetPowerEMS := -100; 
				END_IF 
				IF NOT bSurplusAvailable AND Lynus_Standards.GVL_Energy.stDataOfBatteryInverters[diNrOfEMS_OUT,liLPSetPercentPower].byPriority = bySmGrActiveCommonPrio AND Lynus_Standards.GVL_Energy.stDataOfBatteryInverters[diNrOfEMS_OUT,liLPSetPercentPower].rTargetPowerEMS < 0 THEN 
					Lynus_Standards.GVL_Energy.stDataOfBatteryInverters[diNrOfEMS_OUT,liLPSetPercentPower].rTargetPowerEMS := Lynus_Standards.GVL_Energy.stDataOfBatteryInverters[diNrOfEMS_OUT,liLPSetPercentPower].rTargetPowerEMS + rValuePercentToControllableDevices;
				
				END_IF
				IF NOT bSurplusAvailable AND Lynus_Standards.GVL_Energy.stDataOfBatteryInverters[diNrOfEMS_OUT,liLPSetPercentPower].rTargetPowerEMS > 0 THEN 
					Lynus_Standards.GVL_Energy.stDataOfBatteryInverters[diNrOfEMS_OUT,liLPSetPercentPower].rTargetPowerEMS := 0;
					
				END_IF
				//Power Data is Missing
				IF bMissingPowerData AND Lynus_Standards.GVL_Energy.stDataOfBatteryInverters[diNrOfEMS_OUT,liLPSetPercentPower].byPriority = bySmGrActiveCommonPrio THEN 
					Lynus_Standards.GVL_Energy.stDataOfBatteryInverters[diNrOfEMS_OUT,liLPSetPercentPower].rTargetPowerEMS := 0;	
				END_IF 
				//Limit
							Lynus_Standards.GVL_Energy.stDataOfBatteryInverters[diNrOfEMS_OUT,liLPSetPercentPower].rTargetPowerEMS := LIMIT(-100,Lynus_Standards.GVL_Energy.stDataOfBatteryInverters[diNrOfEMS_OUT,liLPSetPercentPower].rTargetPowerEMS,100);	
			END_FOR
		END_IF
			//Heating pumps
			IF arrActualStepInTurn[1] >= 1 AND arrActualStepInTurn[1] <= 2 THEN
				FOR liLPSetPercentPower := 1 TO Constants_Energy.diMaxNumberOfHeatingPumps BY 1 DO
					//On/Off
					IF bSurplusAvailable AND Lynus_Standards.GVL_Energy.stDataHeatingPumps[diNrOfEMS_OUT,liLPSetPercentPower].byPriority = bySmGrActiveCommonPrio AND Lynus_Standards.GVL_Energy.stDataHeatingPumps[diNrOfEMS_OUT,liLPSetPercentPower].arrTargetPowerEMS[arrActualStepInTurn[1]] < 100 AND NOT 
						Lynus_Standards.GVL_Energy.stDataHeatingPumps[diNrOfEMS_OUT,liLPSetPercentPower].bIsControllable AND NOT Lynus_Standards.GVL_Energy.stDataHeatingPumps[diNrOfEMS_OUT,liLPSetPercentPower].bIsStepSwitched THEN
							Lynus_Standards.GVL_Energy.stDataHeatingPumps[diNrOfEMS_OUT,liLPSetPercentPower].arrTargetPowerEMS[arrActualStepInTurn[1]] := rValuePercentToStepSwitchedDevices; 
					END_IF
					//Controllable linear
					IF bSurplusAvailable AND Lynus_Standards.GVL_Energy.stDataHeatingPumps[diNrOfEMS_OUT,liLPSetPercentPower].byPriority = bySmGrActiveCommonPrio AND Lynus_Standards.GVL_Energy.stDataHeatingPumps[diNrOfEMS_OUT,liLPSetPercentPower].arrTargetPowerEMS[arrActualStepInTurn[1]] < 100 AND 
						Lynus_Standards.GVL_Energy.stDataHeatingPumps[diNrOfEMS_OUT,liLPSetPercentPower].bIsControllable AND NOT Lynus_Standards.GVL_Energy.stDataHeatingPumps[diNrOfEMS_OUT,liLPSetPercentPower].bIsStepSwitched THEN
							Lynus_Standards.GVL_Energy.stDataHeatingPumps[diNrOfEMS_OUT,liLPSetPercentPower].arrTargetPowerEMS[arrActualStepInTurn[1]] := Lynus_Standards.GVL_Energy.stDataHeatingPumps[diNrOfEMS_OUT,liLPSetPercentPower].arrTargetPowerEMS[arrActualStepInTurn[1]] + rValuePercentToControllableDevices; 
					END_IF
					//Step switched
					IF bSurplusAvailable AND Lynus_Standards.GVL_Energy.stDataHeatingPumps[diNrOfEMS_OUT,liLPSetPercentPower].byPriority = bySmGrActiveCommonPrio AND Lynus_Standards.GVL_Energy.stDataHeatingPumps[diNrOfEMS_OUT,liLPSetPercentPower].arrTargetPowerEMS[arrActualStepInTurn[1]] < 100 AND 
						Lynus_Standards.GVL_Energy.stDataHeatingPumps[diNrOfEMS_OUT,liLPSetPercentPower].bIsControllable AND Lynus_Standards.GVL_Energy.stDataHeatingPumps[diNrOfEMS_OUT,liLPSetPercentPower].bIsStepSwitched THEN
							Lynus_Standards.GVL_Energy.stDataHeatingPumps[diNrOfEMS_OUT,liLPSetPercentPower].arrTargetPowerEMS[arrActualStepInTurn[1]] := rValuePercentToStepSwitchedDevices; 
					END_IF
					IF bSurplusAvailable AND Lynus_Standards.GVL_Energy.stDataHeatingPumps[diNrOfEMS_OUT,liLPSetPercentPower].arrTargetPowerEMS[arrActualStepInTurn[1]] > 100 THEN Lynus_Standards.GVL_Energy.stDataHeatingPumps[diNrOfEMS_OUT,liLPSetPercentPower].arrTargetPowerEMS[arrActualStepInTurn[1]] := 100; END_IF 
						//On/Off
						IF NOT bSurplusAvailable AND Lynus_Standards.GVL_Energy.stDataHeatingPumps[diNrOfEMS_OUT,liLPSetPercentPower].byPriority = bySmGrActiveCommonPrio AND Lynus_Standards.GVL_Energy.stDataHeatingPumps[diNrOfEMS_OUT,liLPSetPercentPower].arrTargetPowerEMS[arrActualStepInTurn[1]] > 0 AND NOT 
							Lynus_Standards.GVL_Energy.stDataHeatingPumps[diNrOfEMS_OUT,liLPSetPercentPower].bIsControllable AND NOT Lynus_Standards.GVL_Energy.stDataHeatingPumps[diNrOfEMS_OUT,liLPSetPercentPower].bIsStepSwitched THEN
								Lynus_Standards.GVL_Energy.stDataHeatingPumps[diNrOfEMS_OUT,liLPSetPercentPower].arrTargetPowerEMS[arrActualStepInTurn[1]] := rValuePercentToStepSwitchedDevices; 
						END_IF
						//Controllable linear
						IF NOT bSurplusAvailable AND Lynus_Standards.GVL_Energy.stDataHeatingPumps[diNrOfEMS_OUT,liLPSetPercentPower].byPriority = bySmGrActiveCommonPrio AND Lynus_Standards.GVL_Energy.stDataHeatingPumps[diNrOfEMS_OUT,liLPSetPercentPower].arrTargetPowerEMS[arrActualStepInTurn[1]] > 0 AND 
							Lynus_Standards.GVL_Energy.stDataHeatingPumps[diNrOfEMS_OUT,liLPSetPercentPower].bIsControllable AND NOT Lynus_Standards.GVL_Energy.stDataHeatingPumps[diNrOfEMS_OUT,liLPSetPercentPower].bIsStepSwitched THEN
								Lynus_Standards.GVL_Energy.stDataHeatingPumps[diNrOfEMS_OUT,liLPSetPercentPower].arrTargetPowerEMS[arrActualStepInTurn[1]] := Lynus_Standards.GVL_Energy.stDataHeatingPumps[diNrOfEMS_OUT,liLPSetPercentPower].arrTargetPowerEMS[arrActualStepInTurn[1]] - rValuePercentToControllableDevices; 
						END_IF
						//Step switched
						IF NOT bSurplusAvailable AND Lynus_Standards.GVL_Energy.stDataHeatingPumps[diNrOfEMS_OUT,liLPSetPercentPower].byPriority = bySmGrActiveCommonPrio AND Lynus_Standards.GVL_Energy.stDataHeatingPumps[diNrOfEMS_OUT,liLPSetPercentPower].arrTargetPowerEMS[arrActualStepInTurn[1]] > 0 AND 
							Lynus_Standards.GVL_Energy.stDataHeatingPumps[diNrOfEMS_OUT,liLPSetPercentPower].bIsControllable AND Lynus_Standards.GVL_Energy.stDataHeatingPumps[diNrOfEMS_OUT,liLPSetPercentPower].bIsStepSwitched THEN
								Lynus_Standards.GVL_Energy.stDataHeatingPumps[diNrOfEMS_OUT,liLPSetPercentPower].arrTargetPowerEMS[arrActualStepInTurn[1]] := rValuePercentToStepSwitchedDevices; 
						END_IF
						IF NOT bSurplusAvailable AND Lynus_Standards.GVL_Energy.stDataHeatingPumps[diNrOfEMS_OUT,liLPSetPercentPower].arrTargetPowerEMS[arrActualStepInTurn[1]] < 0 THEN Lynus_Standards.GVL_Energy.stDataHeatingPumps[diNrOfEMS_OUT,liLPSetPercentPower].arrTargetPowerEMS[arrActualStepInTurn[1]] := 0; END_IF
							//Limit
							Lynus_Standards.GVL_Energy.stDataHeatingPumps[diNrOfEMS_OUT,liLPSetPercentPower].arrTargetPowerEMS[arrActualStepInTurn[1]] := LIMIT(0,Lynus_Standards.GVL_Energy.stDataHeatingPumps[diNrOfEMS_OUT,liLPSetPercentPower].arrTargetPowerEMS[arrActualStepInTurn[1]],100);
				END_FOR
			END_IF
				//electric heating element
				IF arrActualStepInTurn[2] >= 1 AND arrActualStepInTurn[2] <= 10 THEN
					FOR liLPSetPercentPower := 1 TO Constants_Energy.diMaxNumberOfElectricHeatingElements BY 1 DO
						//On/Off
						IF bSurplusAvailable AND Lynus_Standards.GVL_Energy.stDataElectricHeatingElements[diNrOfEMS_OUT,liLPSetPercentPower].byPriority = bySmGrActiveCommonPrio AND Lynus_Standards.GVL_Energy.stDataElectricHeatingElements[diNrOfEMS_OUT,liLPSetPercentPower].arrTargetPowerEMS[arrActualStepInTurn[2]] < 100 AND NOT
							Lynus_Standards.GVL_Energy.stDataElectricHeatingElements[diNrOfEMS_OUT,liLPSetPercentPower].bIsControllable AND NOT Lynus_Standards.GVL_Energy.stDataElectricHeatingElements[diNrOfEMS_OUT,liLPSetPercentPower].bIsStepSwitched THEN
								Lynus_Standards.GVL_Energy.stDataElectricHeatingElements[diNrOfEMS_OUT,liLPSetPercentPower].arrTargetPowerEMS[arrActualStepInTurn[2]] := rValuePercentToStepSwitchedDevices;
						END_IF
						//Controllable linear
						IF bSurplusAvailable AND Lynus_Standards.GVL_Energy.stDataElectricHeatingElements[diNrOfEMS_OUT,liLPSetPercentPower].byPriority = bySmGrActiveCommonPrio AND Lynus_Standards.GVL_Energy.stDataElectricHeatingElements[diNrOfEMS_OUT,liLPSetPercentPower].arrTargetPowerEMS[arrActualStepInTurn[2]] < 100 AND
							Lynus_Standards.GVL_Energy.stDataElectricHeatingElements[diNrOfEMS_OUT,liLPSetPercentPower].bIsControllable AND NOT Lynus_Standards.GVL_Energy.stDataElectricHeatingElements[diNrOfEMS_OUT,liLPSetPercentPower].bIsStepSwitched THEN
								Lynus_Standards.GVL_Energy.stDataElectricHeatingElements[diNrOfEMS_OUT,liLPSetPercentPower].arrTargetPowerEMS[arrActualStepInTurn[2]] := Lynus_Standards.GVL_Energy.stDataElectricHeatingElements[diNrOfEMS_OUT,liLPSetPercentPower].arrTargetPowerEMS[arrActualStepInTurn[2]] + rValuePercentToControllableDevices;
						END_IF
						//Step switched
						IF bSurplusAvailable AND Lynus_Standards.GVL_Energy.stDataElectricHeatingElements[diNrOfEMS_OUT,liLPSetPercentPower].byPriority = bySmGrActiveCommonPrio AND Lynus_Standards.GVL_Energy.stDataElectricHeatingElements[diNrOfEMS_OUT,liLPSetPercentPower].arrTargetPowerEMS[arrActualStepInTurn[2]] < 100 AND
							Lynus_Standards.GVL_Energy.stDataElectricHeatingElements[diNrOfEMS_OUT,liLPSetPercentPower].bIsControllable AND Lynus_Standards.GVL_Energy.stDataElectricHeatingElements[diNrOfEMS_OUT,liLPSetPercentPower].bIsStepSwitched THEN
								Lynus_Standards.GVL_Energy.stDataElectricHeatingElements[diNrOfEMS_OUT,liLPSetPercentPower].arrTargetPowerEMS[arrActualStepInTurn[2]] := rValuePercentToStepSwitchedDevices;
						END_IF
						IF bSurplusAvailable AND Lynus_Standards.GVL_Energy.stDataElectricHeatingElements[diNrOfEMS_OUT,liLPSetPercentPower].arrTargetPowerEMS[arrActualStepInTurn[2]] > 100 THEN Lynus_Standards.GVL_Energy.stDataElectricHeatingElements[diNrOfEMS_OUT,liLPSetPercentPower].arrTargetPowerEMS[arrActualStepInTurn[2]] := 100; END_IF
							//On/Off
							IF NOT bSurplusAvailable AND Lynus_Standards.GVL_Energy.stDataElectricHeatingElements[diNrOfEMS_OUT,liLPSetPercentPower].byPriority = bySmGrActiveCommonPrio AND Lynus_Standards.GVL_Energy.stDataElectricHeatingElements[diNrOfEMS_OUT,liLPSetPercentPower].arrTargetPowerEMS[arrActualStepInTurn[2]] > 0 AND NOT
								Lynus_Standards.GVL_Energy.stDataElectricHeatingElements[diNrOfEMS_OUT,liLPSetPercentPower].bIsControllable AND NOT Lynus_Standards.GVL_Energy.stDataElectricHeatingElements[diNrOfEMS_OUT,liLPSetPercentPower].bIsStepSwitched THEN
									Lynus_Standards.GVL_Energy.stDataElectricHeatingElements[diNrOfEMS_OUT,liLPSetPercentPower].arrTargetPowerEMS[arrActualStepInTurn[2]] := rValuePercentToStepSwitchedDevices;
							END_IF
							//Controllable linear
							IF NOT bSurplusAvailable AND Lynus_Standards.GVL_Energy.stDataElectricHeatingElements[diNrOfEMS_OUT,liLPSetPercentPower].byPriority = bySmGrActiveCommonPrio AND Lynus_Standards.GVL_Energy.stDataElectricHeatingElements[diNrOfEMS_OUT,liLPSetPercentPower].arrTargetPowerEMS[arrActualStepInTurn[2]] > 0 AND
								Lynus_Standards.GVL_Energy.stDataElectricHeatingElements[diNrOfEMS_OUT,liLPSetPercentPower].bIsControllable AND NOT Lynus_Standards.GVL_Energy.stDataElectricHeatingElements[diNrOfEMS_OUT,liLPSetPercentPower].bIsStepSwitched THEN
									Lynus_Standards.GVL_Energy.stDataElectricHeatingElements[diNrOfEMS_OUT,liLPSetPercentPower].arrTargetPowerEMS[arrActualStepInTurn[2]] := Lynus_Standards.GVL_Energy.stDataElectricHeatingElements[diNrOfEMS_OUT,liLPSetPercentPower].arrTargetPowerEMS[arrActualStepInTurn[2]] - rValuePercentToControllableDevices;
							END_IF
							//Step switched
							IF NOT bSurplusAvailable AND Lynus_Standards.GVL_Energy.stDataElectricHeatingElements[diNrOfEMS_OUT,liLPSetPercentPower].byPriority = bySmGrActiveCommonPrio AND Lynus_Standards.GVL_Energy.stDataElectricHeatingElements[diNrOfEMS_OUT,liLPSetPercentPower].arrTargetPowerEMS[arrActualStepInTurn[2]] > 0 AND
								Lynus_Standards.GVL_Energy.stDataElectricHeatingElements[diNrOfEMS_OUT,liLPSetPercentPower].bIsControllable AND Lynus_Standards.GVL_Energy.stDataElectricHeatingElements[diNrOfEMS_OUT,liLPSetPercentPower].bIsStepSwitched THEN
									Lynus_Standards.GVL_Energy.stDataElectricHeatingElements[diNrOfEMS_OUT,liLPSetPercentPower].arrTargetPowerEMS[arrActualStepInTurn[2]] := rValuePercentToStepSwitchedDevices;
							END_IF	
							IF NOT bSurplusAvailable AND Lynus_Standards.GVL_Energy.stDataElectricHeatingElements[diNrOfEMS_OUT,liLPSetPercentPower].arrTargetPowerEMS[arrActualStepInTurn[2]] < 0 THEN Lynus_Standards.GVL_Energy.stDataElectricHeatingElements[diNrOfEMS_OUT,liLPSetPercentPower].arrTargetPowerEMS[arrActualStepInTurn[2]] := 0; END_IF 
								//Limit
								Lynus_Standards.GVL_Energy.stDataElectricHeatingElements[diNrOfEMS_OUT,liLPSetPercentPower].arrTargetPowerEMS[arrActualStepInTurn[2]] := LIMIT(0,Lynus_Standards.GVL_Energy.stDataElectricHeatingElements[diNrOfEMS_OUT,liLPSetPercentPower].arrTargetPowerEMS[arrActualStepInTurn[2]],100);
					END_FOR			
				END_IF
					//Other big consumer
					FOR liLPSetPercentPower := 1 TO Constants_Energy.diMaxNumberOfOtherBigConsumers BY 1 DO
						//On/Off
						IF bSurplusAvailable AND Lynus_Standards.GVL_Energy.stDataOtherBigConsumers[diNrOfEMS_OUT,liLPSetPercentPower].byPriority = bySmGrActiveCommonPrio AND Lynus_Standards.GVL_Energy.stDataOtherBigConsumers[diNrOfEMS_OUT,liLPSetPercentPower].rTargetPowerEMS < 100 AND NOT
							Lynus_Standards.GVL_Energy.stDataOtherBigConsumers[diNrOfEMS_OUT,liLPSetPercentPower].bIsControllable THEN Lynus_Standards.GVL_Energy.stDataOtherBigConsumers[diNrOfEMS_OUT,liLPSetPercentPower].rTargetPowerEMS := rValuePercentToStepSwitchedDevices; 
						END_IF
						//Controllable linear
						IF bSurplusAvailable AND Lynus_Standards.GVL_Energy.stDataOtherBigConsumers[diNrOfEMS_OUT,liLPSetPercentPower].byPriority = bySmGrActiveCommonPrio AND Lynus_Standards.GVL_Energy.stDataOtherBigConsumers[diNrOfEMS_OUT,liLPSetPercentPower].rTargetPowerEMS < 100 AND
							Lynus_Standards.GVL_Energy.stDataOtherBigConsumers[diNrOfEMS_OUT,liLPSetPercentPower].bIsControllable THEN Lynus_Standards.GVL_Energy.stDataOtherBigConsumers[diNrOfEMS_OUT,liLPSetPercentPower].rTargetPowerEMS := Lynus_Standards.GVL_Energy.stDataOtherBigConsumers[diNrOfEMS_OUT,liLPSetPercentPower].rTargetPowerEMS + rValuePercentToControllableDevices;
						END_IF
						IF bSurplusAvailable AND Lynus_Standards.GVL_Energy.stDataOtherBigConsumers[diNrOfEMS_OUT,liLPSetPercentPower].rTargetPowerEMS > 100 THEN Lynus_Standards.GVL_Energy.stDataOtherBigConsumers[diNrOfEMS_OUT,liLPSetPercentPower].rTargetPowerEMS := 100; END_IF
							//On/Off
							IF NOT bSurplusAvailable AND Lynus_Standards.GVL_Energy.stDataOtherBigConsumers[diNrOfEMS_OUT,liLPSetPercentPower].byPriority = bySmGrActiveCommonPrio AND Lynus_Standards.GVL_Energy.stDataOtherBigConsumers[diNrOfEMS_OUT,liLPSetPercentPower].rTargetPowerEMS > 0 AND NOT
								Lynus_Standards.GVL_Energy.stDataOtherBigConsumers[diNrOfEMS_OUT,liLPSetPercentPower].bIsControllable THEN Lynus_Standards.GVL_Energy.stDataOtherBigConsumers[diNrOfEMS_OUT,liLPSetPercentPower].rTargetPowerEMS := rValuePercentToStepSwitchedDevices; 
							END_IF
							//Controllable linear
							IF NOT bSurplusAvailable AND Lynus_Standards.GVL_Energy.stDataOtherBigConsumers[diNrOfEMS_OUT,liLPSetPercentPower].byPriority = bySmGrActiveCommonPrio AND Lynus_Standards.GVL_Energy.stDataOtherBigConsumers[diNrOfEMS_OUT,liLPSetPercentPower].rTargetPowerEMS > 0 AND
								Lynus_Standards.GVL_Energy.stDataOtherBigConsumers[diNrOfEMS_OUT,liLPSetPercentPower].bIsControllable THEN Lynus_Standards.GVL_Energy.stDataOtherBigConsumers[diNrOfEMS_OUT,liLPSetPercentPower].rTargetPowerEMS := Lynus_Standards.GVL_Energy.stDataOtherBigConsumers[diNrOfEMS_OUT,liLPSetPercentPower].rTargetPowerEMS - rValuePercentToControllableDevices;
							END_IF
							IF NOT bSurplusAvailable AND Lynus_Standards.GVL_Energy.stDataOtherBigConsumers[diNrOfEMS_OUT,liLPSetPercentPower].rTargetPowerEMS < 0 THEN Lynus_Standards.GVL_Energy.stDataOtherBigConsumers[diNrOfEMS_OUT,liLPSetPercentPower].rTargetPowerEMS := 0; END_IF
								//Limit
								Lynus_Standards.GVL_Energy.stDataOtherBigConsumers[diNrOfEMS_OUT,liLPSetPercentPower].rTargetPowerEMS := LIMIT(0,Lynus_Standards.GVL_Energy.stDataOtherBigConsumers[diNrOfEMS_OUT,liLPSetPercentPower].rTargetPowerEMS,100);
					END_FOR
						//Electric charging stations
						FOR liLPSetPercentPower := 1 TO Constants_Energy.diMaxNumberOfElectricChargingStations BY 1 DO
							//On/Off
							IF bSurplusAvailable AND Lynus_Standards.GVL_Energy.stDataElectricChargingStations[diNrOfEMS_OUT,liLPSetPercentPower].byPriority = bySmGrActiveCommonPrio AND Lynus_Standards.GVL_Energy.stDataElectricChargingStations[diNrOfEMS_OUT,liLPSetPercentPower].rTargetPowerEMS < 100 AND NOT 
								Lynus_Standards.GVL_Energy.stDataElectricChargingStations[diNrOfEMS_OUT,liLPSetPercentPower].bIsControllable THEN 
									//No power on ECS because on the Electric Fuse Line we take to much Power on witch the ECS is conected
									IF NOT bNoPowerForECS THEN 
										Lynus_Standards.GVL_Energy.stDataElectricChargingStations[diNrOfEMS_OUT,liLPSetPercentPower].rTargetPowerEMS := rValuePercentToStepSwitchedDevices;	
									END_IF	
							END_IF
							//Controllable linear
							IF bSurplusAvailable AND Lynus_Standards.GVL_Energy.stDataElectricChargingStations[diNrOfEMS_OUT,liLPSetPercentPower].byPriority = bySmGrActiveCommonPrio AND Lynus_Standards.GVL_Energy.stDataElectricChargingStations[diNrOfEMS_OUT,liLPSetPercentPower].rTargetPowerEMS < 100 AND 
								Lynus_Standards.GVL_Energy.stDataElectricChargingStations[diNrOfEMS_OUT,liLPSetPercentPower].bIsControllable THEN 
									//No power on ECS because on the Electric Fuse Line we take to much Power on witch the ECS is conected
									IF NOT bNoPowerForECS THEN
										Lynus_Standards.GVL_Energy.stDataElectricChargingStations[diNrOfEMS_OUT,liLPSetPercentPower].rTargetPowerEMS := Lynus_Standards.GVL_Energy.stDataElectricChargingStations[diNrOfEMS_OUT,liLPSetPercentPower].rTargetPowerEMS + rValuePercentToControllableDevices;		
									END_IF
							END_IF
							IF bSurplusAvailable AND Lynus_Standards.GVL_Energy.stDataElectricChargingStations[diNrOfEMS_OUT,liLPSetPercentPower].rTargetPowerEMS > 100 THEN Lynus_Standards.GVL_Energy.stDataElectricChargingStations[diNrOfEMS_OUT,liLPSetPercentPower].rTargetPowerEMS := 100; END_IF
								//On/Off
								IF NOT bSurplusAvailable AND Lynus_Standards.GVL_Energy.stDataElectricChargingStations[diNrOfEMS_OUT,liLPSetPercentPower].byPriority = bySmGrActiveCommonPrio AND Lynus_Standards.GVL_Energy.stDataElectricChargingStations[diNrOfEMS_OUT,liLPSetPercentPower].rTargetPowerEMS > 0 AND NOT 
									Lynus_Standards.GVL_Energy.stDataElectricChargingStations[diNrOfEMS_OUT,liLPSetPercentPower].bIsControllable THEN Lynus_Standards.GVL_Energy.stDataElectricChargingStations[diNrOfEMS_OUT,liLPSetPercentPower].rTargetPowerEMS := rValuePercentToStepSwitchedDevices;		
								END_IF
								//Controllable linear
								IF NOT bSurplusAvailable AND Lynus_Standards.GVL_Energy.stDataElectricChargingStations[diNrOfEMS_OUT,liLPSetPercentPower].byPriority = bySmGrActiveCommonPrio AND Lynus_Standards.GVL_Energy.stDataElectricChargingStations[diNrOfEMS_OUT,liLPSetPercentPower].rTargetPowerEMS > 0 AND 
									Lynus_Standards.GVL_Energy.stDataElectricChargingStations[diNrOfEMS_OUT,liLPSetPercentPower].bIsControllable THEN Lynus_Standards.GVL_Energy.stDataElectricChargingStations[diNrOfEMS_OUT,liLPSetPercentPower].rTargetPowerEMS := Lynus_Standards.GVL_Energy.stDataElectricChargingStations[diNrOfEMS_OUT,liLPSetPercentPower].rTargetPowerEMS - rValuePercentToControllableDevices;		
								END_IF
								IF NOT bSurplusAvailable AND Lynus_Standards.GVL_Energy.stDataElectricChargingStations[diNrOfEMS_OUT,liLPSetPercentPower].rTargetPowerEMS < 0 THEN Lynus_Standards.GVL_Energy.stDataElectricChargingStations[diNrOfEMS_OUT,liLPSetPercentPower].rTargetPowerEMS := 0; END_IF	
									//Limit
									Lynus_Standards.GVL_Energy.stDataElectricChargingStations[diNrOfEMS_OUT,liLPSetPercentPower].rTargetPowerEMS := LIMIT(0,Lynus_Standards.GVL_Energy.stDataElectricChargingStations[diNrOfEMS_OUT,liLPSetPercentPower].rTargetPowerEMS,100);
						END_FOR 
		uiState := 10;
END_CASE

(*-------------------------------------------------------------------------------------Correction Charging stations regarding max fuse power---------------------------------------------------------------------------------------------------------------*)

//Correction for the charging station power that the target power is not bigger then the maximum of the fuse. Active on mode peak load capping (Index from meter > 0 and fuse value > 0) and load management (always).
//Work only with controllable charging station. Not work for On/off stations.
IF (stSetupEMS.bEnableMainFuseFunction AND bEnable AND (eOperationMode = E_OperatingMode_EMS.ePeakLoadCapping OR eOperationMode = E_OperatingMode_EMS.eLoadManagement)) THEN

IF arrMaxPrioReached[5] THEN bECSPrio255 := TRUE; END_IF
	IF NOT bSurplusAvailable THEN bECSPrio255 := FALSE; END_IF

lrPowerDiffFuseECS := (stSetupEMS.rSizeMainFuseCS * 0.95) - Lynus_Standards.GVL_Energy.stDataElectricMeters[diNrOfEM_IN_ECS].lrPowerConsumption;	
	//Make little tolerance that we dont regulate up and down 
	IF lrPowerDiffFuseECS > 0 AND lrPowerDiffFuseECS <= 0.1 THEN lrPowerDiffFuseECS := 0; END_IF  
		IF lrPowerDiffFuseECS > 0 THEN lrPowerDiffFuseECS := lrPowerDiffFuseECS - 0.1; END_IF 
	
	//No power for ECS on normal EMS Step
	IF lrPowerDiffFuseECS < 0 THEN 
		bNoPowerForECS := TRUE; 
	ELSE
		bNoPowerForECS := FALSE;
	END_IF	
		
	diNumberOfECS := 0;		
		FOR liLPCorrectionPowerCS := 1 TO Constants_Energy.diMaxNumberOfElectricChargingStations BY 1 DO
			//Count number of charging stations when we have surplus on Fuse Line
			IF NOT arrMinPrioReached[5] AND Lynus_Standards.GVL_Energy.stDataElectricChargingStations[diNrOfEMS_OUT,liLPCorrectionPowerCS].byPriority <= bySmGrActiveCommonPrio AND 
				Lynus_Standards.GVL_Energy.stDataElectricChargingStations[diNrOfEMS_OUT,liLPCorrectionPowerCS].bEnabled AND 
					Lynus_Standards.GVL_Energy.stDataElectricChargingStations[diNrOfEMS_OUT,liLPCorrectionPowerCS].rTargetPowerEMS < 100 AND lrPowerDiffFuseECS >= 0 THEN 
						diNumberOfECS := diNumberOfECS + 1; 
			END_IF
				//Count number of charging stations when we have NO surplus on Fuse Line
				IF NOT arrMinPrioReached[5] AND Lynus_Standards.GVL_Energy.stDataElectricChargingStations[diNrOfEMS_OUT,liLPCorrectionPowerCS].byPriority <= bySmGrActiveCommonPrio AND 
					Lynus_Standards.GVL_Energy.stDataElectricChargingStations[diNrOfEMS_OUT,liLPCorrectionPowerCS].bEnabled AND
						Lynus_Standards.GVL_Energy.stDataElectricChargingStations[diNrOfEMS_OUT,liLPCorrectionPowerCS].rTargetPowerEMS > 0 AND lrPowerDiffFuseECS < 0 THEN 
							diNumberOfECS := diNumberOfECS + 1; 
				END_IF 
		END_FOR
			//Calculate the power in % for each charging station
			//Actual Power is <= then stSetupEMS.rSizeMainFuseCS 
			IF diNumberOfECS > 0 AND lrPowerDiffFuseECS >= 0 THEN lrPowerForCalculateECS := lrPowerDiffFuseECS / diNumberOfECS; END_IF  
				//Actual Power is > then stSetupEMS.rSizeMainFuseCS
				IF diNumberOfECS > 0 AND lrPowerDiffFuseECS < 0 THEN lrPowerForCalculateECS := (lrPowerDiffFuseECS * - 1) / diNumberOfECS; END_IF 

//Timer to make the correction for the charging stations
IF (NOT arrMinPrioReached[5] AND NOT timCorrectionECS.Q AND bEnable AND (eOperationMode = E_OperatingMode_EMS.ePeakLoadCapping OR eOperationMode = E_OperatingMode_EMS.eLoadManagement)) THEN  
	timCorrectionECS.IN := TRUE;
ELSE
	timCorrectionECS.IN := FALSE;
END_IF
	//The timer work faster when the value from lrPowerDiffFuseECS is bigger
	//Positive value (Mean more power for ECS)
	IF lrPowerDiffFuseECS >= 0.75 THEN timCorrectionECS.PT := T#2.5S; END_IF
	IF lrPowerDiffFuseECS >= 0.5 AND lrPowerDiffFuseECS < 0.75 THEN timCorrectionECS.PT := T#3S; END_IF
	IF lrPowerDiffFuseECS >= 0.25 AND lrPowerDiffFuseECS < 0.5 THEN timCorrectionECS.PT := T#3.5S; END_IF
	IF lrPowerDiffFuseECS > 0 AND lrPowerDiffFuseECS < 0.25 THEN timCorrectionECS.PT := T#4S; END_IF
		//Value is 0
		IF lrPowerDiffFuseECS = 0 THEN timCorrectionECS.PT := T#5S; END_IF 
			//Negative value (Mean less power for ECS)
			IF lrPowerDiffFuseECS < 0 AND lrPowerDiffFuseECS > - 0.25 THEN timCorrectionECS.PT := T#4S; END_IF
			IF lrPowerDiffFuseECS <= - 0.25 AND lrPowerDiffFuseECS > - 0.5 THEN timCorrectionECS.PT := T#3.5S; END_IF
			IF lrPowerDiffFuseECS <= - 0.5 AND lrPowerDiffFuseECS > - 0.75 THEN timCorrectionECS.PT := T#3S; END_IF
			IF lrPowerDiffFuseECS <= - 0.75 THEN timCorrectionECS.PT := T#2.5S; END_IF
				//Timer
				timCorrectionECS(IN:= , PT:= , Q=> , ET=> );				
				
//Set the new power to the charging stations with priority < common priority in progress
lrTargetPowerCorrectionECS := 0;
	FOR liLPCorrectionPowerCS := 1 TO Constants_Energy.diMaxNumberOfElectricChargingStations BY 1 DO 	
		IF (NOT arrMinPrioReached[5] AND timCorrectionECS.Q AND Lynus_Standards.GVL_Energy.stDataElectricChargingStations[diNrOfEMS_OUT,liLPCorrectionPowerCS].byPriority < bySmGrActiveCommonPrio AND eOperationMode = E_OperatingMode_EMS.ePeakLoadCapping AND stSetupEMS.rSizeMainFuseCS > 0 AND Lynus_Standards.GVL_Energy.stDataElectricMeters[diNrOfEM_IN_ECS].bEnabled) OR
			(NOT arrMinPrioReached[5] AND timCorrectionECS.Q AND Lynus_Standards.GVL_Energy.stDataElectricChargingStations[diNrOfEMS_OUT,liLPCorrectionPowerCS].byPriority < bySmGrActiveCommonPrio AND eOperationMode = E_OperatingMode_EMS.eLoadManagement AND stSetupEMS.rSizeMainFuseCS > 0 AND Lynus_Standards.GVL_Energy.stDataElectricMeters[diNrOfEM_IN_ECS].bEnabled) OR
				(NOT arrMinPrioReached[5] AND timCorrectionECS.Q AND lrPowerDiffFuseECS < 0 AND Lynus_Standards.GVL_Energy.stDataElectricChargingStations[diNrOfEMS_OUT,liLPCorrectionPowerCS].byPriority = bySmGrActiveCommonPrio AND eOperationMode = E_OperatingMode_EMS.ePeakLoadCapping AND stSetupEMS.rSizeMainFuseCS > 0 AND Lynus_Standards.GVL_Energy.stDataElectricMeters[diNrOfEM_IN_ECS].bEnabled) OR
				(NOT arrMinPrioReached[5] AND timCorrectionECS.Q AND lrPowerDiffFuseECS < 0 AND Lynus_Standards.GVL_Energy.stDataElectricChargingStations[diNrOfEMS_OUT,liLPCorrectionPowerCS].byPriority = bySmGrActiveCommonPrio AND eOperationMode = E_OperatingMode_EMS.eLoadManagement AND stSetupEMS.rSizeMainFuseCS > 0 AND Lynus_Standards.GVL_Energy.stDataElectricMeters[diNrOfEM_IN_ECS].bEnabled) OR				
					(NOT arrMinPrioReached[5] AND timCorrectionECS.Q AND Lynus_Standards.GVL_Energy.stDataElectricChargingStations[diNrOfEMS_OUT,liLPCorrectionPowerCS].byPriority = 255 AND bECSPrio255 AND eOperationMode = E_OperatingMode_EMS.ePeakLoadCapping AND stSetupEMS.rSizeMainFuseCS > 0 AND Lynus_Standards.GVL_Energy.stDataElectricMeters[diNrOfEM_IN_ECS].bEnabled) OR	
					(NOT arrMinPrioReached[5] AND timCorrectionECS.Q AND Lynus_Standards.GVL_Energy.stDataElectricChargingStations[diNrOfEMS_OUT,liLPCorrectionPowerCS].byPriority = 255 AND bECSPrio255 AND eOperationMode = E_OperatingMode_EMS.eLoadManagement AND stSetupEMS.rSizeMainFuseCS > 0 AND Lynus_Standards.GVL_Energy.stDataElectricMeters[diNrOfEM_IN_ECS].bEnabled) THEN
						//Calcualte the new % value for each charging station	
						IF Lynus_Standards.GVL_Energy.stDataElectricChargingStations[diNrOfEMS_OUT,liLPCorrectionPowerCS].rMaxPower > 0 THEN 
							lrTargetPowerCorrectionECS := (100 * lrPowerForCalculateECS) / Lynus_Standards.GVL_Energy.stDataElectricChargingStations[diNrOfEMS_OUT,liLPCorrectionPowerCS].rMaxPower;	
								lrTargetPowerCorrectionECS := LIMIT(0,lrTargetPowerCorrectionECS,100);
						ELSE
							//Without power data on the setups from the charging station set target powert to -100 or +100 to dissable the charging station
							IF lrPowerDiffFuseECS >= 0 THEN lrTargetPowerCorrectionECS := - 100; ELSE lrTargetPowerCorrectionECS := 100; END_IF 
						END_IF	
							IF lrPowerDiffFuseECS >= 0 AND Lynus_Standards.GVL_Energy.stDataElectricChargingStations[diNrOfEMS_OUT,liLPCorrectionPowerCS].bIsControllable THEN 
								Lynus_Standards.GVL_Energy.stDataElectricChargingStations[diNrOfEMS_OUT,liLPCorrectionPowerCS].rTargetPowerEMS := Lynus_Standards.GVL_Energy.stDataElectricChargingStations[diNrOfEMS_OUT,liLPCorrectionPowerCS].rTargetPowerEMS + LREAL_TO_REAL(lrTargetPowerCorrectionECS); 
							END_IF
								IF lrPowerDiffFuseECS < 0 AND Lynus_Standards.GVL_Energy.stDataElectricChargingStations[diNrOfEMS_OUT,liLPCorrectionPowerCS].bIsControllable THEN 
									Lynus_Standards.GVL_Energy.stDataElectricChargingStations[diNrOfEMS_OUT,liLPCorrectionPowerCS].rTargetPowerEMS := Lynus_Standards.GVL_Energy.stDataElectricChargingStations[diNrOfEMS_OUT,liLPCorrectionPowerCS].rTargetPowerEMS - LREAL_TO_REAL(lrTargetPowerCorrectionECS); 
								END_IF	
									//Limits
									Lynus_Standards.GVL_Energy.stDataElectricChargingStations[diNrOfEMS_OUT,liLPCorrectionPowerCS].rTargetPowerEMS := LIMIT(0,Lynus_Standards.GVL_Energy.stDataElectricChargingStations[diNrOfEMS_OUT,liLPCorrectionPowerCS].rTargetPowerEMS,100);			
		END_IF
	END_FOR

//Dissable the ECS complete when the EM has a Error
IF (Lynus_Standards.GVL_Energy.stDataElectricMeters[diNrOfEM_IN_ECS].byErrorWarning = 2 AND (eOperationMode = E_OperatingMode_EMS.eLoadManagement OR eOperationMode = E_OperatingMode_EMS.ePeakLoadCapping)) THEN
	timResetDisableECS.IN := TRUE;
ELSE
	timResetDisableECS.IN := FALSE;
END_IF
	timResetDisableECS(IN:= , PT:= T#10S, Q=> , ET=> );	
		IF timResetDisableECS.Q THEN bDisableECS := TRUE; ELSE bDisableECS := FALSE; END_IF

ELSE
	timResetDisableECS.IN := FALSE;
		bDisableECS := FALSE;		
			timCorrectionECS.IN := FALSE;
				bECSPrio255 := FALSE;
					bNoPowerForECS := FALSE;
END_IF		
		
(*-------------------------------------------------------------------------------------Set the power to 0 on each device---------------------------------------------------------------------------------------------------------------*)	
	
//When a device has the priority 0, the priority is bigger then who was at the moment in progress, the EMS function is not enabled, a positv or negative edge came when the emergency power mode start or stop or when the operation mode is changing then the EMS start from new and all devices are set to defaul target power 0.
//Set the target power to 0 where there should no power 

FPEPO(CLK:= bEPMActive, Q=> );
	FNEPO(CLK:= bEPMActive, Q=> );
	
diMemCmpOperationState := MEMCMP(ADR(eOperationMode),ADR(eOperationModeEMS_CP),SIZEOF(eOperationModeEMS_CP)); 	

//Battery	
FOR arrLPPrioZeroSetToZeroP[1] := 1 TO Constants_Energy.diMaxNumberOfBatteryInverters BY 1 DO
	IF Lynus_Standards.GVL_Energy.stDataOfBatteryInverters[diNrOfEMS_OUT,arrLPPrioZeroSetToZeroP[1]].byPriority = 0 OR Lynus_Standards.GVL_Energy.stDataOfBatteryInverters[diNrOfEMS_OUT,arrLPPrioZeroSetToZeroP[1]].byPriority > arrActualPrioInTurn[1] OR arrMinPrioReached[1] OR NOT bEnable OR FPEPO.Q OR FNEPO.Q OR 
		diMemCmpOperationState <> 0 OR eOperationMode = E_OperatingMode_EMS.eAllOff OR bStopAll THEN 
			Lynus_Standards.GVL_Energy.stDataOfBatteryInverters[diNrOfEMS_OUT,arrLPPrioZeroSetToZeroP[1]].rTargetPowerEMS := 0; 
	END_IF
END_FOR
	//Heating Pumps
	FOR arrLPPrioZeroSetToZeroP[2] := 1 TO Constants_Energy.diMaxNumberOfHeatingPumps BY 1 DO
		IF Lynus_Standards.GVL_Energy.stDataHeatingPumps[diNrOfEMS_OUT,arrLPPrioZeroSetToZeroP[2]].byPriority = 0 OR Lynus_Standards.GVL_Energy.stDataHeatingPumps[diNrOfEMS_OUT,arrLPPrioZeroSetToZeroP[2]].byPriority > arrActualPrioInTurn[2] OR arrMinPrioReached[2] OR NOT bEnable OR FPEPO.Q OR FNEPO.Q OR 
			diMemCmpOperationState <> 0 OR eOperationMode = E_OperatingMode_EMS.eAllOff OR bStopAll THEN
				Lynus_Standards.GVL_Energy.stDataHeatingPumps[diNrOfEMS_OUT,arrLPPrioZeroSetToZeroP[2]].arrTargetPowerEMS[1] := 0;
					Lynus_Standards.GVL_Energy.stDataHeatingPumps[diNrOfEMS_OUT,arrLPPrioZeroSetToZeroP[2]].arrTargetPowerEMS[2] := 0;
						//Switch off external on command for heating pumps
						Lynus_Standards.GVL_Energy.stDataHeatingPumps[diNrOfEMS_OUT,arrLPPrioZeroSetToZeroP[2]].bExternalOnCommand := FALSE;
		END_IF
	END_FOR
		//EHE
		FOR arrLPPrioZeroSetToZeroP[3] := 1 TO Constants_Energy.diMaxNumberOfElectricHeatingElements BY 1 DO
			IF Lynus_Standards.GVL_Energy.stDataElectricHeatingElements[diNrOfEMS_OUT,arrLPPrioZeroSetToZeroP[3]].byPriority = 0 OR Lynus_Standards.GVL_Energy.stDataElectricHeatingElements[diNrOfEMS_OUT,arrLPPrioZeroSetToZeroP[3]].byPriority > arrActualPrioInTurn[3] OR arrMinPrioReached[3] OR NOT bEnable OR FPEPO.Q OR FNEPO.Q OR 
				diMemCmpOperationState <> 0 OR eOperationMode = E_OperatingMode_EMS.eAllOff OR bStopAll THEN 
					Lynus_Standards.GVL_Energy.stDataElectricHeatingElements[diNrOfEMS_OUT,arrLPPrioZeroSetToZeroP[3]].arrTargetPowerEMS[1] := 0;
						Lynus_Standards.GVL_Energy.stDataElectricHeatingElements[diNrOfEMS_OUT,arrLPPrioZeroSetToZeroP[3]].arrTargetPowerEMS[2] := 0;
							Lynus_Standards.GVL_Energy.stDataElectricHeatingElements[diNrOfEMS_OUT,arrLPPrioZeroSetToZeroP[3]].arrTargetPowerEMS[3] := 0;
								Lynus_Standards.GVL_Energy.stDataElectricHeatingElements[diNrOfEMS_OUT,arrLPPrioZeroSetToZeroP[3]].arrTargetPowerEMS[4] := 0;
									Lynus_Standards.GVL_Energy.stDataElectricHeatingElements[diNrOfEMS_OUT,arrLPPrioZeroSetToZeroP[3]].arrTargetPowerEMS[5] := 0;
					Lynus_Standards.GVL_Energy.stDataElectricHeatingElements[diNrOfEMS_OUT,arrLPPrioZeroSetToZeroP[3]].arrTargetPowerEMS[6] := 0;
						Lynus_Standards.GVL_Energy.stDataElectricHeatingElements[diNrOfEMS_OUT,arrLPPrioZeroSetToZeroP[3]].arrTargetPowerEMS[7] := 0;
							Lynus_Standards.GVL_Energy.stDataElectricHeatingElements[diNrOfEMS_OUT,arrLPPrioZeroSetToZeroP[3]].arrTargetPowerEMS[8] := 0;
								Lynus_Standards.GVL_Energy.stDataElectricHeatingElements[diNrOfEMS_OUT,arrLPPrioZeroSetToZeroP[3]].arrTargetPowerEMS[9] := 0;
									Lynus_Standards.GVL_Energy.stDataElectricHeatingElements[diNrOfEMS_OUT,arrLPPrioZeroSetToZeroP[3]].arrTargetPowerEMS[10] := 0;
			END_IF
		END_FOR
			//OBC
			FOR arrLPPrioZeroSetToZeroP[4] := 1 TO Constants_Energy.diMaxNumberOfOtherBigConsumers BY 1 DO
				IF Lynus_Standards.GVL_Energy.stDataOtherBigConsumers[diNrOfEMS_OUT,arrLPPrioZeroSetToZeroP[4]].byPriority = 0 OR Lynus_Standards.GVL_Energy.stDataOtherBigConsumers[diNrOfEMS_OUT,arrLPPrioZeroSetToZeroP[4]].byPriority > arrActualPrioInTurn[4] OR arrMinPrioReached[4] OR NOT bEnable OR FPEPO.Q OR 
					FNEPO.Q OR diMemCmpOperationState <> 0 OR eOperationMode = E_OperatingMode_EMS.eAllOff OR bStopAll THEN
						Lynus_Standards.GVL_Energy.stDataOtherBigConsumers[diNrOfEMS_OUT,arrLPPrioZeroSetToZeroP[4]].rTargetPowerEMS := 0;
				END_IF
			END_FOR
				//ECS
				FOR arrLPPrioZeroSetToZeroP[5] := 1 TO Constants_Energy.diMaxNumberOfElectricChargingStations BY 1 DO
					IF Lynus_Standards.GVL_Energy.stDataElectricChargingStations[diNrOfEMS_OUT,arrLPPrioZeroSetToZeroP[5]].byPriority = 0 OR Lynus_Standards.GVL_Energy.stDataElectricChargingStations[diNrOfEMS_OUT,arrLPPrioZeroSetToZeroP[5]].byPriority > arrActualPrioInTurn[5] OR arrMinPrioReached[5] OR NOT bEnable OR FPEPO.Q OR FNEPO.Q OR 
						diMemCmpOperationState <> 0 OR eOperationMode = E_OperatingMode_EMS.eAllOff OR bStopAll OR 
							((eOperationMode = E_OperatingMode_EMS.ePeakLoadCapping OR eOperationMode = E_OperatingMode_EMS.eLoadManagement) AND stSetupEMS.bEnableMainFuseFunction AND (NOT Lynus_Standards.GVL_Energy.stDataElectricMeters[diNrOfEM_IN_ECS].bEnabled OR stSetupEMS.rSizeMainFuseCS <= 0 OR bDisableECS)) THEN
								Lynus_Standards.GVL_Energy.stDataElectricChargingStations[diNrOfEMS_OUT,arrLPPrioZeroSetToZeroP[5]].rTargetPowerEMS := 0;
					END_IF
				END_FOR

(*----------------------------------------------------------------------------------------------------Controller to discharge/charge the batterys on the different modes----------------------------------------------------------------------------------------------------------*)
(*----------------------------------------------------------------------------------------------------Controller to discharge the battery in the self consumption mode----------------------------------------------------------------------------------------------------------*)

lrErrorPIDCorrectionBattSC := ABS(0 - lrGridPower);

//Controller weighting
IF eSpeedModeLocalController = E_SpeedModeLocalController_EMS.eSlow THEN 
	IF lrErrorPIDCorrectionBattSC <= 0.5 THEN fbPIDBatterySC.rPValue := 0.05; fbPIDBatterySC.udiIValue := 450;
	ELSIF lrErrorPIDCorrectionBattSC > 0.5 AND lrErrorPIDCorrectionBattSC <= 1 THEN fbPIDBatterySC.rPValue := 0.07; fbPIDBatterySC.udiIValue := 450;
	ELSIF lrErrorPIDCorrectionBattSC > 1 AND lrErrorPIDCorrectionBattSC <= 1.5 THEN fbPIDBatterySC.rPValue := 0.09; fbPIDBatterySC.udiIValue := 450; 
	ELSIF lrErrorPIDCorrectionBattSC > 1.5 AND lrErrorPIDCorrectionBattSC <= 2 THEN fbPIDBatterySC.rPValue := 0.11; fbPIDBatterySC.udiIValue := 450; 	
	ELSIF lrErrorPIDCorrectionBattSC > 2 AND lrErrorPIDCorrectionBattSC <= 2.5 THEN fbPIDBatterySC.rPValue := 0.13; fbPIDBatterySC.udiIValue := 675; 
	ELSIF lrErrorPIDCorrectionBattSC > 2.5 AND lrErrorPIDCorrectionBattSC <= 3 THEN fbPIDBatterySC.rPValue := 0.15; fbPIDBatterySC.udiIValue := 675;
	ELSIF lrErrorPIDCorrectionBattSC > 3 AND lrErrorPIDCorrectionBattSC <= 3.5 THEN fbPIDBatterySC.rPValue := 0.17; fbPIDBatterySC.udiIValue := 900;
	ELSIF lrErrorPIDCorrectionBattSC > 3.5 AND lrErrorPIDCorrectionBattSC <= 4 THEN fbPIDBatterySC.rPValue := 0.19; fbPIDBatterySC.udiIValue := 900;
	ELSIF lrErrorPIDCorrectionBattSC > 4 AND lrErrorPIDCorrectionBattSC <= 4.5 THEN fbPIDBatterySC.rPValue := 0.21; fbPIDBatterySC.udiIValue := 900;
	ELSIF lrErrorPIDCorrectionBattSC > 4.5 AND lrErrorPIDCorrectionBattSC <= 5 THEN fbPIDBatterySC.rPValue := 0.23; fbPIDBatterySC.udiIValue := 900;
	ELSIF lrErrorPIDCorrectionBattSC > 5 THEN fbPIDBatterySC.rPValue := 0.25; fbPIDBatterySC.udiIValue := 900;
	END_IF
ELSIF eSpeedModeLocalController = E_SpeedModeLocalController_EMS.eBalanced THEN 
	IF lrErrorPIDCorrectionBattSC <= 0.5 THEN fbPIDBatterySC.rPValue := 0.10; fbPIDBatterySC.udiIValue := 450;
	ELSIF lrErrorPIDCorrectionBattSC > 0.5 AND lrErrorPIDCorrectionBattSC <= 1 THEN fbPIDBatterySC.rPValue := 0.14; fbPIDBatterySC.udiIValue := 450;
	ELSIF lrErrorPIDCorrectionBattSC > 1 AND lrErrorPIDCorrectionBattSC <= 1.5 THEN fbPIDBatterySC.rPValue := 0.18; fbPIDBatterySC.udiIValue := 450; 
	ELSIF lrErrorPIDCorrectionBattSC > 1.5 AND lrErrorPIDCorrectionBattSC <= 2 THEN fbPIDBatterySC.rPValue := 0.22; fbPIDBatterySC.udiIValue := 450; 	
	ELSIF lrErrorPIDCorrectionBattSC > 2 AND lrErrorPIDCorrectionBattSC <= 2.5 THEN fbPIDBatterySC.rPValue := 0.26; fbPIDBatterySC.udiIValue := 675; 
	ELSIF lrErrorPIDCorrectionBattSC > 2.5 AND lrErrorPIDCorrectionBattSC <= 3 THEN fbPIDBatterySC.rPValue := 0.30; fbPIDBatterySC.udiIValue := 675;
	ELSIF lrErrorPIDCorrectionBattSC > 3 AND lrErrorPIDCorrectionBattSC <= 3.5 THEN fbPIDBatterySC.rPValue := 0.34; fbPIDBatterySC.udiIValue := 900;
	ELSIF lrErrorPIDCorrectionBattSC > 3.5 AND lrErrorPIDCorrectionBattSC <= 4 THEN fbPIDBatterySC.rPValue := 0.38; fbPIDBatterySC.udiIValue := 900;
	ELSIF lrErrorPIDCorrectionBattSC > 4 AND lrErrorPIDCorrectionBattSC <= 4.5 THEN fbPIDBatterySC.rPValue := 0.42; fbPIDBatterySC.udiIValue := 900;
	ELSIF lrErrorPIDCorrectionBattSC > 4.5 AND lrErrorPIDCorrectionBattSC <= 5 THEN fbPIDBatterySC.rPValue := 0.46; fbPIDBatterySC.udiIValue := 900;
	ELSIF lrErrorPIDCorrectionBattSC > 5 THEN fbPIDBatterySC.rPValue := 0.50; fbPIDBatterySC.udiIValue := 900;
	END_IF
ELSIF eSpeedModeLocalController = E_SpeedModeLocalController_EMS.eFast THEN
	IF lrErrorPIDCorrectionBattSC <= 0.5 THEN fbPIDBatterySC.rPValue := 0.30; fbPIDBatterySC.udiIValue := 275;
	ELSIF lrErrorPIDCorrectionBattSC > 0.5 AND lrErrorPIDCorrectionBattSC <= 1 THEN fbPIDBatterySC.rPValue := 0.33; fbPIDBatterySC.udiIValue := 275;
	ELSIF lrErrorPIDCorrectionBattSC > 1 AND lrErrorPIDCorrectionBattSC <= 1.5 THEN fbPIDBatterySC.rPValue := 0.36; fbPIDBatterySC.udiIValue := 275; 
	ELSIF lrErrorPIDCorrectionBattSC > 1.5 AND lrErrorPIDCorrectionBattSC <= 2 THEN fbPIDBatterySC.rPValue := 0.39; fbPIDBatterySC.udiIValue := 275; 	
	ELSIF lrErrorPIDCorrectionBattSC > 2 AND lrErrorPIDCorrectionBattSC <= 2.5 THEN fbPIDBatterySC.rPValue := 0.42; fbPIDBatterySC.udiIValue := 500; 
	ELSIF lrErrorPIDCorrectionBattSC > 2.5 AND lrErrorPIDCorrectionBattSC <= 3 THEN fbPIDBatterySC.rPValue := 0.45; fbPIDBatterySC.udiIValue := 500;
	ELSIF lrErrorPIDCorrectionBattSC > 3 AND lrErrorPIDCorrectionBattSC <= 3.5 THEN fbPIDBatterySC.rPValue := 0.48; fbPIDBatterySC.udiIValue := 750;
	ELSIF lrErrorPIDCorrectionBattSC > 3.5 AND lrErrorPIDCorrectionBattSC <= 4 THEN fbPIDBatterySC.rPValue := 0.51; fbPIDBatterySC.udiIValue := 750;
	ELSIF lrErrorPIDCorrectionBattSC > 4 AND lrErrorPIDCorrectionBattSC <= 4.5 THEN fbPIDBatterySC.rPValue := 0.54; fbPIDBatterySC.udiIValue := 750;
	ELSIF lrErrorPIDCorrectionBattSC > 4.5 AND lrErrorPIDCorrectionBattSC <= 5 THEN fbPIDBatterySC.rPValue := 0.57; fbPIDBatterySC.udiIValue := 750;
	ELSIF lrErrorPIDCorrectionBattSC > 5 THEN fbPIDBatterySC.rPValue := 0.60; fbPIDBatterySC.udiIValue := 750;
	END_IF
END_IF

IF bEnable AND eOperationMode = E_OperatingMode_EMS.eSelfConsumption AND NOT bEPMActive AND NOT bStopAll AND NOT bDischrgCmdFromBackendOK AND 
	arrMinPrioReached[1] AND arrMinPrioReached[2] AND arrMinPrioReached[3] AND arrMinPrioReached[4] AND arrMinPrioReached[5] THEN
		fbPIDBatterySC.bEnable := TRUE;
ELSE
		fbPIDBatterySC.bEnable := FALSE;
END_IF

fbPIDBatterySC( 
	bEnable:= , 
	rSetpoint:= 0, 
	udiIValue:= , 
	udiDValue:= 0, 
	udiDamping:= 0, 
	rPValue:= , 
	rMaxValue:= 100, 
	rMinValue:= 0, 
	rNeutralZone:= 0.1, 
	bDirection:= TRUE, 
	rActualValue:= LREAL_TO_REAL(lrGridPower), 
	rQController=> rControllerQPIDSC);

//Set the Controller output	to 0 when we have surplus. (Because its possible that the controller output is not set 100% to 0 regarding internal discrepancies)
IF rControllerQPIDSC <= 0.4 AND fbPIDBatterySC.bEnable AND lrGridPower <= - Constants_Energy.rToleranceSurplusConsumption THEN 
	timPIDSC.IN := TRUE;
ELSE
	timPIDSC.IN := FALSE;
END_IF

timPIDSC(IN:= , PT:= T#15S, Q=> , ET=> );
	IF timPIDSC.Q THEN rControllerQPIDSC := 0; END_IF	

FOR liLPDataBatteryInverter := 1 TO Constants_Energy.diMaxNumberOfBatteryInverters BY 1 DO
	IF Lynus_Standards.GVL_Energy.stDataOfBatteryInverters[diNrOfEMS_OUT,liLPDataBatteryInverter].byPriority <> 0 AND NOT bEPMActive AND eOperationMode = E_OperatingMode_EMS.eSelfConsumption AND	
		arrMinPrioReached[1] AND arrMinPrioReached[2] AND arrMinPrioReached[3] AND arrMinPrioReached[4] AND arrMinPrioReached[5] THEN
			Lynus_Standards.GVL_Energy.stDataOfBatteryInverters[diNrOfEMS_OUT,liLPDataBatteryInverter].rTargetPowerEMS := rControllerQPIDSC;
	END_IF 
END_FOR	

(*----------------------------------------------------------------------------------------------------Controller to charge and discharge the battery in the peak load capping mode and load management mode----------------------------------------------------------------------------------------------------------*)

//IMPORTANT : On this 2 modes the Batterys are allways active.
//This means that in these two modes the battery is not processed via the state machine like other devices.
//They are there to limit the power to the grid connection. The batteries charge according to the release when the power on the grid is below the grid connection or when power is fed back to the grid.
//The 95% are used so that the remaining 5% are still seen as surplus and thus the remaining consumers can still be regulated up to take advantage of the full grid connection.
//The batteries are processed with their priorities during charging. THIS means that only those batteries are active which also match the current active priority in the EMS.

(*--------------------------------------------------------------------------------------------------------------------Discharge the batterys-----------------------------------------------------------------------------------------------------------------------------------------------*)

lrErrorPIDCorrectionBattPLCLM_Dischrg := ABS(lrGridPower - (lrSizeGridConnection * 0.95));

//Controller weighting
IF eSpeedModeLocalController = E_SpeedModeLocalController_EMS.eSlow THEN 
	IF lrErrorPIDCorrectionBattPLCLM_Dischrg <= 0.5 THEN fbPIDBatteryPLCLM_Dischrg.rPValue := 0.05; fbPIDBatteryPLCLM_Dischrg.udiIValue := 450;
	ELSIF lrErrorPIDCorrectionBattPLCLM_Dischrg > 0.5 AND lrErrorPIDCorrectionBattPLCLM_Dischrg <= 1 THEN fbPIDBatteryPLCLM_Dischrg.rPValue := 0.07; fbPIDBatteryPLCLM_Dischrg.udiIValue := 450;
	ELSIF lrErrorPIDCorrectionBattPLCLM_Dischrg > 1 AND lrErrorPIDCorrectionBattPLCLM_Dischrg <= 1.5 THEN fbPIDBatteryPLCLM_Dischrg.rPValue := 0.09; fbPIDBatteryPLCLM_Dischrg.udiIValue := 450; 
	ELSIF lrErrorPIDCorrectionBattPLCLM_Dischrg > 1.5 AND lrErrorPIDCorrectionBattPLCLM_Dischrg <= 2 THEN fbPIDBatteryPLCLM_Dischrg.rPValue := 0.11; fbPIDBatteryPLCLM_Dischrg.udiIValue := 450; 	
	ELSIF lrErrorPIDCorrectionBattPLCLM_Dischrg > 2 AND lrErrorPIDCorrectionBattPLCLM_Dischrg <= 2.5 THEN fbPIDBatteryPLCLM_Dischrg.rPValue := 0.13; fbPIDBatteryPLCLM_Dischrg.udiIValue := 675; 
	ELSIF lrErrorPIDCorrectionBattPLCLM_Dischrg > 2.5 AND lrErrorPIDCorrectionBattPLCLM_Dischrg <= 3 THEN fbPIDBatteryPLCLM_Dischrg.rPValue := 0.15; fbPIDBatteryPLCLM_Dischrg.udiIValue := 675;
	ELSIF lrErrorPIDCorrectionBattPLCLM_Dischrg > 3 AND lrErrorPIDCorrectionBattPLCLM_Dischrg <= 3.5 THEN fbPIDBatteryPLCLM_Dischrg.rPValue := 0.17; fbPIDBatteryPLCLM_Dischrg.udiIValue := 900;
	ELSIF lrErrorPIDCorrectionBattPLCLM_Dischrg > 3.5 AND lrErrorPIDCorrectionBattPLCLM_Dischrg <= 4 THEN fbPIDBatteryPLCLM_Dischrg.rPValue := 0.19; fbPIDBatteryPLCLM_Dischrg.udiIValue := 900;
	ELSIF lrErrorPIDCorrectionBattPLCLM_Dischrg > 4 AND lrErrorPIDCorrectionBattPLCLM_Dischrg <= 4.5 THEN fbPIDBatteryPLCLM_Dischrg.rPValue := 0.21; fbPIDBatteryPLCLM_Dischrg.udiIValue := 900;
	ELSIF lrErrorPIDCorrectionBattPLCLM_Dischrg > 4.5 AND lrErrorPIDCorrectionBattPLCLM_Dischrg <= 5 THEN fbPIDBatteryPLCLM_Dischrg.rPValue := 0.23; fbPIDBatteryPLCLM_Dischrg.udiIValue := 900;
	ELSIF lrErrorPIDCorrectionBattPLCLM_Dischrg > 5 THEN fbPIDBatteryPLCLM_Dischrg.rPValue := 0.25; fbPIDBatteryPLCLM_Dischrg.udiIValue := 900;
	END_IF
ELSIF eSpeedModeLocalController = E_SpeedModeLocalController_EMS.eBalanced THEN
	IF lrErrorPIDCorrectionBattPLCLM_Dischrg <= 0.5 THEN fbPIDBatteryPLCLM_Dischrg.rPValue := 0.10; fbPIDBatteryPLCLM_Dischrg.udiIValue := 450;
	ELSIF lrErrorPIDCorrectionBattPLCLM_Dischrg > 0.5 AND lrErrorPIDCorrectionBattPLCLM_Dischrg <= 1 THEN fbPIDBatteryPLCLM_Dischrg.rPValue := 0.14; fbPIDBatteryPLCLM_Dischrg.udiIValue := 450;
	ELSIF lrErrorPIDCorrectionBattPLCLM_Dischrg > 1 AND lrErrorPIDCorrectionBattPLCLM_Dischrg <= 1.5 THEN fbPIDBatteryPLCLM_Dischrg.rPValue := 0.18; fbPIDBatteryPLCLM_Dischrg.udiIValue := 450; 
	ELSIF lrErrorPIDCorrectionBattPLCLM_Dischrg > 1.5 AND lrErrorPIDCorrectionBattPLCLM_Dischrg <= 2 THEN fbPIDBatteryPLCLM_Dischrg.rPValue := 0.22; fbPIDBatteryPLCLM_Dischrg.udiIValue := 450; 	
	ELSIF lrErrorPIDCorrectionBattPLCLM_Dischrg > 2 AND lrErrorPIDCorrectionBattPLCLM_Dischrg <= 2.5 THEN fbPIDBatteryPLCLM_Dischrg.rPValue := 0.26; fbPIDBatteryPLCLM_Dischrg.udiIValue := 675; 
	ELSIF lrErrorPIDCorrectionBattPLCLM_Dischrg > 2.5 AND lrErrorPIDCorrectionBattPLCLM_Dischrg <= 3 THEN fbPIDBatteryPLCLM_Dischrg.rPValue := 0.30; fbPIDBatteryPLCLM_Dischrg.udiIValue := 675;
	ELSIF lrErrorPIDCorrectionBattPLCLM_Dischrg > 3 AND lrErrorPIDCorrectionBattPLCLM_Dischrg <= 3.5 THEN fbPIDBatteryPLCLM_Dischrg.rPValue := 0.34; fbPIDBatteryPLCLM_Dischrg.udiIValue := 900;
	ELSIF lrErrorPIDCorrectionBattPLCLM_Dischrg > 3.5 AND lrErrorPIDCorrectionBattPLCLM_Dischrg <= 4 THEN fbPIDBatteryPLCLM_Dischrg.rPValue := 0.38; fbPIDBatteryPLCLM_Dischrg.udiIValue := 900;
	ELSIF lrErrorPIDCorrectionBattPLCLM_Dischrg > 4 AND lrErrorPIDCorrectionBattPLCLM_Dischrg <= 4.5 THEN fbPIDBatteryPLCLM_Dischrg.rPValue := 0.42; fbPIDBatteryPLCLM_Dischrg.udiIValue := 900;
	ELSIF lrErrorPIDCorrectionBattPLCLM_Dischrg > 4.5 AND lrErrorPIDCorrectionBattPLCLM_Dischrg <= 5 THEN fbPIDBatteryPLCLM_Dischrg.rPValue := 0.46; fbPIDBatteryPLCLM_Dischrg.udiIValue := 900;
	ELSIF lrErrorPIDCorrectionBattPLCLM_Dischrg > 5 THEN fbPIDBatteryPLCLM_Dischrg.rPValue := 0.50; fbPIDBatteryPLCLM_Dischrg.udiIValue := 900;
	END_IF
ELSIF eSpeedModeLocalController = E_SpeedModeLocalController_EMS.eFast THEN
	IF lrErrorPIDCorrectionBattPLCLM_Dischrg <= 0.5 THEN fbPIDBatteryPLCLM_Dischrg.rPValue := 0.30; fbPIDBatteryPLCLM_Dischrg.udiIValue := 275;
	ELSIF lrErrorPIDCorrectionBattPLCLM_Dischrg > 0.5 AND lrErrorPIDCorrectionBattPLCLM_Dischrg <= 1 THEN fbPIDBatteryPLCLM_Dischrg.rPValue := 0.33; fbPIDBatteryPLCLM_Dischrg.udiIValue := 275;
	ELSIF lrErrorPIDCorrectionBattPLCLM_Dischrg > 1 AND lrErrorPIDCorrectionBattPLCLM_Dischrg <= 1.5 THEN fbPIDBatteryPLCLM_Dischrg.rPValue := 0.36; fbPIDBatteryPLCLM_Dischrg.udiIValue := 275; 
	ELSIF lrErrorPIDCorrectionBattPLCLM_Dischrg > 1.5 AND lrErrorPIDCorrectionBattPLCLM_Dischrg <= 2 THEN fbPIDBatteryPLCLM_Dischrg.rPValue := 0.39; fbPIDBatteryPLCLM_Dischrg.udiIValue := 275; 	
	ELSIF lrErrorPIDCorrectionBattPLCLM_Dischrg > 2 AND lrErrorPIDCorrectionBattPLCLM_Dischrg <= 2.5 THEN fbPIDBatteryPLCLM_Dischrg.rPValue := 0.42; fbPIDBatteryPLCLM_Dischrg.udiIValue := 500; 
	ELSIF lrErrorPIDCorrectionBattPLCLM_Dischrg > 2.5 AND lrErrorPIDCorrectionBattPLCLM_Dischrg <= 3 THEN fbPIDBatteryPLCLM_Dischrg.rPValue := 0.45; fbPIDBatteryPLCLM_Dischrg.udiIValue := 500;
	ELSIF lrErrorPIDCorrectionBattPLCLM_Dischrg > 3 AND lrErrorPIDCorrectionBattPLCLM_Dischrg <= 3.5 THEN fbPIDBatteryPLCLM_Dischrg.rPValue := 0.48; fbPIDBatteryPLCLM_Dischrg.udiIValue := 750;
	ELSIF lrErrorPIDCorrectionBattPLCLM_Dischrg > 3.5 AND lrErrorPIDCorrectionBattPLCLM_Dischrg <= 4 THEN fbPIDBatteryPLCLM_Dischrg.rPValue := 0.51; fbPIDBatteryPLCLM_Dischrg.udiIValue := 750;
	ELSIF lrErrorPIDCorrectionBattPLCLM_Dischrg > 4 AND lrErrorPIDCorrectionBattPLCLM_Dischrg <= 4.5 THEN fbPIDBatteryPLCLM_Dischrg.rPValue := 0.54; fbPIDBatteryPLCLM_Dischrg.udiIValue := 750;
	ELSIF lrErrorPIDCorrectionBattPLCLM_Dischrg > 4.5 AND lrErrorPIDCorrectionBattPLCLM_Dischrg <= 5 THEN fbPIDBatteryPLCLM_Dischrg.rPValue := 0.57; fbPIDBatteryPLCLM_Dischrg.udiIValue := 750;
	ELSIF lrErrorPIDCorrectionBattPLCLM_Dischrg > 5 THEN fbPIDBatteryPLCLM_Dischrg.rPValue := 0.60; fbPIDBatteryPLCLM_Dischrg.udiIValue := 750;
	END_IF
END_IF 

IF (bEnable AND eOperationMode = E_OperatingMode_EMS.ePeakLoadCapping AND NOT bEPMActive AND NOT bStopAll AND NOT bDischrgCmdFromBackendOK AND NOT fbPIDBatteryPLCLM_Chrg.bEnable AND lrGridPower >= (lrSizeGridConnection * 0.95)) OR 
	(bEnable AND eOperationMode = E_OperatingMode_EMS.eLoadManagement AND NOT bEPMActive AND NOT bStopAll AND NOT bDischrgCmdFromBackendOK AND NOT fbPIDBatteryPLCLM_Chrg.bEnable AND lrGridPower >= (SEL(b_ZeroPowerRegulation,lrSizeGridConnection,0) * 0.95)) THEN				
		fbPIDBatteryPLCLM_Dischrg.bEnable := TRUE;
END_IF
	IF NOT bEnable OR diNumberOfActiveBatterys = 0 OR bEPMActive OR bStopAll OR bDischrgCmdFromBackendOK OR fbPIDBatteryPLCLM_Chrg.bEnable OR eOperationMode = E_OperatingMode_EMS.eAllOff OR eOperationMode = E_OperatingMode_EMS.eSelfConsumption OR
		(lrGridPower < (SEL(b_ZeroPowerRegulation,lrSizeGridConnection,0) * 0.95) AND fbPIDBatteryPLCLM_Dischrg.rQController <= 0) THEN
		fbPIDBatteryPLCLM_Dischrg.bEnable := FALSE;
	END_IF    

fbPIDBatteryPLCLM_Dischrg( 
	bEnable:= , 
	rSetpoint:= lreal_to_real(SEL(b_ZeroPowerRegulation,lrSizeGridConnection,0)),		
	udiIValue:= , 
	udiDValue:= 0, 
	udiDamping:= 0, 
	rPValue:= , 
	rMaxValue:= 100, 
	rMinValue:= 0, 
	rNeutralZone:= 0.1, 
	bDirection:= TRUE, 
	rActualValue:= LREAL_TO_REAL(lrGridPower), 
	rQController=> );

FOR liLPDataBatteryInverter := 1 TO Constants_Energy.diMaxNumberOfBatteryInverters BY 1 DO
	IF Lynus_Standards.GVL_Energy.stDataOfBatteryInverters[diNrOfEMS_OUT,liLPDataBatteryInverter].byPriority <> 0 AND NOT bEPMActive AND fbPIDBatteryPLCLM_Dischrg.bEnable THEN
		Lynus_Standards.GVL_Energy.stDataOfBatteryInverters[diNrOfEMS_OUT,liLPDataBatteryInverter].rTargetPowerEMS := fbPIDBatteryPLCLM_Dischrg.rQController;
	END_IF 
END_FOR	

(*--------------------------------------------------------------------------------------------------------------------Charge the batterys-----------------------------------------------------------------------------------------------------------------------------------------------*)

IF stSetupEMS.bAllowChrgFromGrid THEN 
	lrErrorPIDCorrectionBattPLCLM_Chrg := ABS(lrGridPower - (lrSizeGridConnection * 0.95));
ELSE
	lrErrorPIDCorrectionBattPLCLM_Chrg := ABS(0 - lrGridPower);
END_IF 

//Controller weighting
IF eSpeedModeLocalController = E_SpeedModeLocalController_EMS.eSlow THEN 
	IF lrErrorPIDCorrectionBattPLCLM_Chrg <= 0.5 THEN fbPIDBatteryPLCLM_Chrg.rPValue := 0.05; fbPIDBatteryPLCLM_Chrg.udiIValue := 450;
	ELSIF lrErrorPIDCorrectionBattPLCLM_Chrg > 0.5 AND lrErrorPIDCorrectionBattPLCLM_Chrg <= 1 THEN fbPIDBatteryPLCLM_Chrg.rPValue := 0.07; fbPIDBatteryPLCLM_Chrg.udiIValue := 450;
	ELSIF lrErrorPIDCorrectionBattPLCLM_Chrg > 1 AND lrErrorPIDCorrectionBattPLCLM_Chrg <= 1.5 THEN fbPIDBatteryPLCLM_Chrg.rPValue := 0.09; fbPIDBatteryPLCLM_Chrg.udiIValue := 450; 
	ELSIF lrErrorPIDCorrectionBattPLCLM_Chrg > 1.5 AND lrErrorPIDCorrectionBattPLCLM_Chrg <= 2 THEN fbPIDBatteryPLCLM_Chrg.rPValue := 0.11; fbPIDBatteryPLCLM_Chrg.udiIValue := 450; 	
	ELSIF lrErrorPIDCorrectionBattPLCLM_Chrg > 2 AND lrErrorPIDCorrectionBattPLCLM_Chrg <= 2.5 THEN fbPIDBatteryPLCLM_Chrg.rPValue := 0.13; fbPIDBatteryPLCLM_Chrg.udiIValue := 675; 
	ELSIF lrErrorPIDCorrectionBattPLCLM_Chrg > 2.5 AND lrErrorPIDCorrectionBattPLCLM_Chrg <= 3 THEN fbPIDBatteryPLCLM_Chrg.rPValue := 0.15; fbPIDBatteryPLCLM_Chrg.udiIValue := 675;
	ELSIF lrErrorPIDCorrectionBattPLCLM_Chrg > 3 AND lrErrorPIDCorrectionBattPLCLM_Chrg <= 3.5 THEN fbPIDBatteryPLCLM_Chrg.rPValue := 0.17; fbPIDBatteryPLCLM_Chrg.udiIValue := 900;
	ELSIF lrErrorPIDCorrectionBattPLCLM_Chrg > 3.5 AND lrErrorPIDCorrectionBattPLCLM_Chrg <= 4 THEN fbPIDBatteryPLCLM_Chrg.rPValue := 0.19; fbPIDBatteryPLCLM_Chrg.udiIValue := 900;
	ELSIF lrErrorPIDCorrectionBattPLCLM_Chrg > 4 AND lrErrorPIDCorrectionBattPLCLM_Chrg <= 4.5 THEN fbPIDBatteryPLCLM_Chrg.rPValue := 0.21; fbPIDBatteryPLCLM_Chrg.udiIValue := 900;
	ELSIF lrErrorPIDCorrectionBattPLCLM_Chrg > 4.5 AND lrErrorPIDCorrectionBattPLCLM_Chrg <= 5 THEN fbPIDBatteryPLCLM_Chrg.rPValue := 0.23; fbPIDBatteryPLCLM_Chrg.udiIValue := 900;
	ELSIF lrErrorPIDCorrectionBattPLCLM_Chrg > 5 THEN fbPIDBatteryPLCLM_Chrg.rPValue := 0.25; fbPIDBatteryPLCLM_Chrg.udiIValue := 900;
	END_IF
ELSIF eSpeedModeLocalController = E_SpeedModeLocalController_EMS.eBalanced THEN
	IF lrErrorPIDCorrectionBattPLCLM_Chrg <= 0.5 THEN fbPIDBatteryPLCLM_Chrg.rPValue := 0.10; fbPIDBatteryPLCLM_Chrg.udiIValue := 450;
	ELSIF lrErrorPIDCorrectionBattPLCLM_Chrg > 0.5 AND lrErrorPIDCorrectionBattPLCLM_Chrg <= 1 THEN fbPIDBatteryPLCLM_Chrg.rPValue := 0.14; fbPIDBatteryPLCLM_Chrg.udiIValue := 450;
	ELSIF lrErrorPIDCorrectionBattPLCLM_Chrg > 1 AND lrErrorPIDCorrectionBattPLCLM_Chrg <= 1.5 THEN fbPIDBatteryPLCLM_Chrg.rPValue := 0.18; fbPIDBatteryPLCLM_Chrg.udiIValue := 450; 
	ELSIF lrErrorPIDCorrectionBattPLCLM_Chrg > 1.5 AND lrErrorPIDCorrectionBattPLCLM_Chrg <= 2 THEN fbPIDBatteryPLCLM_Chrg.rPValue := 0.22; fbPIDBatteryPLCLM_Chrg.udiIValue := 450; 	
	ELSIF lrErrorPIDCorrectionBattPLCLM_Chrg > 2 AND lrErrorPIDCorrectionBattPLCLM_Chrg <= 2.5 THEN fbPIDBatteryPLCLM_Chrg.rPValue := 0.26; fbPIDBatteryPLCLM_Chrg.udiIValue := 675; 
	ELSIF lrErrorPIDCorrectionBattPLCLM_Chrg > 2.5 AND lrErrorPIDCorrectionBattPLCLM_Chrg <= 3 THEN fbPIDBatteryPLCLM_Chrg.rPValue := 0.30; fbPIDBatteryPLCLM_Chrg.udiIValue := 675;
	ELSIF lrErrorPIDCorrectionBattPLCLM_Chrg > 3 AND lrErrorPIDCorrectionBattPLCLM_Chrg <= 3.5 THEN fbPIDBatteryPLCLM_Chrg.rPValue := 0.34; fbPIDBatteryPLCLM_Chrg.udiIValue := 900;
	ELSIF lrErrorPIDCorrectionBattPLCLM_Chrg > 3.5 AND lrErrorPIDCorrectionBattPLCLM_Chrg <= 4 THEN fbPIDBatteryPLCLM_Chrg.rPValue := 0.38; fbPIDBatteryPLCLM_Chrg.udiIValue := 900;
	ELSIF lrErrorPIDCorrectionBattPLCLM_Chrg > 4 AND lrErrorPIDCorrectionBattPLCLM_Chrg <= 4.5 THEN fbPIDBatteryPLCLM_Chrg.rPValue := 0.42; fbPIDBatteryPLCLM_Chrg.udiIValue := 900;
	ELSIF lrErrorPIDCorrectionBattPLCLM_Chrg > 4.5 AND lrErrorPIDCorrectionBattPLCLM_Chrg <= 5 THEN fbPIDBatteryPLCLM_Chrg.rPValue := 0.46; fbPIDBatteryPLCLM_Chrg.udiIValue := 900;
	ELSIF lrErrorPIDCorrectionBattPLCLM_Chrg > 5 THEN fbPIDBatteryPLCLM_Chrg.rPValue := 0.50; fbPIDBatteryPLCLM_Chrg.udiIValue := 900;
	END_IF
ELSIF eSpeedModeLocalController = E_SpeedModeLocalController_EMS.eFast THEN
	IF lrErrorPIDCorrectionBattPLCLM_Chrg <= 0.5 THEN fbPIDBatteryPLCLM_Chrg.rPValue := 0.30; fbPIDBatteryPLCLM_Chrg.udiIValue := 275;
	ELSIF lrErrorPIDCorrectionBattPLCLM_Chrg > 0.5 AND lrErrorPIDCorrectionBattPLCLM_Chrg <= 1 THEN fbPIDBatteryPLCLM_Chrg.rPValue := 0.33; fbPIDBatteryPLCLM_Chrg.udiIValue := 275;
	ELSIF lrErrorPIDCorrectionBattPLCLM_Chrg > 1 AND lrErrorPIDCorrectionBattPLCLM_Chrg <= 1.5 THEN fbPIDBatteryPLCLM_Chrg.rPValue := 0.36; fbPIDBatteryPLCLM_Chrg.udiIValue := 275; 
	ELSIF lrErrorPIDCorrectionBattPLCLM_Chrg > 1.5 AND lrErrorPIDCorrectionBattPLCLM_Chrg <= 2 THEN fbPIDBatteryPLCLM_Chrg.rPValue := 0.39; fbPIDBatteryPLCLM_Chrg.udiIValue := 275; 	
	ELSIF lrErrorPIDCorrectionBattPLCLM_Chrg > 2 AND lrErrorPIDCorrectionBattPLCLM_Chrg <= 2.5 THEN fbPIDBatteryPLCLM_Chrg.rPValue := 0.42; fbPIDBatteryPLCLM_Chrg.udiIValue := 500; 
	ELSIF lrErrorPIDCorrectionBattPLCLM_Chrg > 2.5 AND lrErrorPIDCorrectionBattPLCLM_Chrg <= 3 THEN fbPIDBatteryPLCLM_Chrg.rPValue := 0.45; fbPIDBatteryPLCLM_Chrg.udiIValue := 500;
	ELSIF lrErrorPIDCorrectionBattPLCLM_Chrg > 3 AND lrErrorPIDCorrectionBattPLCLM_Chrg <= 3.5 THEN fbPIDBatteryPLCLM_Chrg.rPValue := 0.48; fbPIDBatteryPLCLM_Chrg.udiIValue := 750;
	ELSIF lrErrorPIDCorrectionBattPLCLM_Chrg > 3.5 AND lrErrorPIDCorrectionBattPLCLM_Chrg <= 4 THEN fbPIDBatteryPLCLM_Chrg.rPValue := 0.51; fbPIDBatteryPLCLM_Chrg.udiIValue := 750;
	ELSIF lrErrorPIDCorrectionBattPLCLM_Chrg > 4 AND lrErrorPIDCorrectionBattPLCLM_Chrg <= 4.5 THEN fbPIDBatteryPLCLM_Chrg.rPValue := 0.54; fbPIDBatteryPLCLM_Chrg.udiIValue := 750;
	ELSIF lrErrorPIDCorrectionBattPLCLM_Chrg > 4.5 AND lrErrorPIDCorrectionBattPLCLM_Chrg <= 5 THEN fbPIDBatteryPLCLM_Chrg.rPValue := 0.57; fbPIDBatteryPLCLM_Chrg.udiIValue := 750;
	ELSIF lrErrorPIDCorrectionBattPLCLM_Chrg > 5 THEN fbPIDBatteryPLCLM_Chrg.rPValue := 0.60; fbPIDBatteryPLCLM_Chrg.udiIValue := 750;
	END_IF	
END_IF

//Start and stop charge when charging from thr grid is allowed
IF (bEnable AND eOperationMode = E_OperatingMode_EMS.ePeakLoadCapping AND stSetupEMS.bAllowChrgFromGrid AND NOT bEPMActive AND NOT bStopAll AND NOT 
		fbPIDBatteryPLCLM_Dischrg.bEnable AND NOT fbPIDDischrgCmdFromBackend.bEnable AND lrGridPower < (lrSizeGridConnection * 0.95)) AND (b_TimeBasedReleaseChargingBattery OR NOT b_EnableBatteryChargingControl) OR 
	(bEnable AND eOperationMode = E_OperatingMode_EMS.eLoadManagement AND stSetupEMS.bAllowChrgFromGrid AND NOT bEPMActive AND NOT bStopAll AND NOT 
		fbPIDBatteryPLCLM_Dischrg.bEnable AND NOT fbPIDDischrgCmdFromBackend.bEnable AND lrGridPower < (lrSizeGridConnection * 0.95)) 
THEN
			fbPIDBatteryPLCLM_Chrg.bEnable := TRUE;
END_IF
	IF (stSetupEMS.bAllowChrgFromGrid AND (NOT bEnable OR diNumberOfActiveBatterys = 0 OR bEPMActive OR bStopAll OR fbPIDBatteryPLCLM_Dischrg.bEnable OR eOperationMode = E_OperatingMode_EMS.eAllOff OR 
		eOperationMode = E_OperatingMode_EMS.eSelfConsumption OR fbPIDDischrgCmdFromBackend.bEnable OR (fbPIDBatteryPLCLM_Chrg.rQController >= 0 AND lrGridPower >= (lrSizeGridConnection * 0.95)))) or not b_TimeBasedReleaseChargingBattery THEN
			fbPIDBatteryPLCLM_Chrg.bEnable := FALSE;
	END_IF

//Start and stop charge when charging from thr grid is not allowed
IF (bEnable AND eOperationMode = E_OperatingMode_EMS.ePeakLoadCapping AND NOT stSetupEMS.bAllowChrgFromGrid AND NOT bEPMActive AND NOT bStopAll AND NOT 
		fbPIDBatteryPLCLM_Dischrg.bEnable AND NOT fbPIDDischrgCmdFromBackend.bEnable AND lrGridPower < 0) OR 
	(bEnable AND eOperationMode = E_OperatingMode_EMS.eLoadManagement AND NOT stSetupEMS.bAllowChrgFromGrid AND NOT bEPMActive AND NOT bStopAll AND NOT 
		fbPIDBatteryPLCLM_Dischrg.bEnable AND NOT fbPIDDischrgCmdFromBackend.bEnable AND lrGridPower < 0) THEN
			fbPIDBatteryPLCLM_Chrg.bEnable := TRUE;
END_IF
	IF (NOT stSetupEMS.bAllowChrgFromGrid AND (NOT bEnable OR diNumberOfActiveBatterys = 0 OR bEPMActive OR bStopAll OR fbPIDBatteryPLCLM_Dischrg.bEnable OR eOperationMode = E_OperatingMode_EMS.eAllOff OR 
		eOperationMode = E_OperatingMode_EMS.eSelfConsumption OR fbPIDDischrgCmdFromBackend.bEnable OR (fbPIDBatteryPLCLM_Chrg.rQController >= 0 AND lrGridPower >= 0))) THEN
			fbPIDBatteryPLCLM_Chrg.bEnable := FALSE;
	END_IF

//Set the Setpoint from the controller	
IF stSetupEMS.bAllowChrgFromGrid AND dwAvarageBatterySOC < stSetupEMS.byResChrgfromGridToBatt THEN 
	fbPIDBatteryPLCLM_Chrg.rSetpoint := LREAL_TO_REAL(lrSizeGridConnection * 0.95);
ELSE
	fbPIDBatteryPLCLM_Chrg.rSetpoint := 0;
END_IF 	
	
